TEXTLIST S4_Alarms
  0 = 'Station 4 Clamp A1 Failed to Advance... Check Q1.0...' | German: 'S4 0 Row 1 Failed To Advance.. Check Qxxx.x German' | French: 'S4 0 Row 1 Failed To Advance.. Check Qxxx.x French' | 汉语: '汉语'
  1 = 'Station 4 Clamp A1 Failed to Return... Check Q1.1...' | German: 'S4 1 Row 1 Failed To Return.. Check Qxxx.x German' | French: 'S4 1 Row 1 Failed To Return.. Check Qxxx.x French' | 汉语: '汉语'
  2 = 'Station 4 Clamp A1 Lost Advanced... Check I1.0...' | German: 'S4 2 Row 1 Lost Advance Position... Check Ixxx.x German' | French: 'S4 2 Row 1 Lost Advance Position... Check Ixxx.x French' | 汉语: '汉语'
  3 = 'Station 4 Clamp A1 Lost Returned... Check I1.1...' | German: 'S4 3 Row 1 Lost Return Position... Check Ixxx.x German' | French: 'S4 3 Row 1 Lost Return Position... Check Ixxx.x French'
  4 = 'Station 4 Clamp A1 Switch Fault... Check I1.0, I1.1...' | German: 'S4 4 Row 1 Switch Fault... Check Ixxx.x / Ixxx.x German' | French: 'S4 4 Row 1 Switch Fault... Check Ixxx.x / Ixxx.x French'
  5 = 'Spare' | German: 'S4 5 Row 1 Spare Message German' | French: 'S4 5 Row 1 Spare Message French'
  6 = 'Spare' | German: 'S4 6 Row 1 Spare Message German' | French: 'S4 6 Row 1 Spare Message French'
  7 = 'Spare' | German: 'S4 7 Row 1 Spare Message German' | French: 'S4 7 Row 1 Spare Message French'
  8 = 'Spare' | German: 'S4 8 Row 1 Spare Message German' | French: 'S4 8 Row 1 Spare Message French'
  9 = 'Spare' | German: 'S4 9 Row 1 Spare Message German' | French: 'S4 9 Row 1 Spare Message French'
  10 = 'Lock Cylinder A2 Failed to Lock... Check Q1.2...' | German: 'S4 10 Row 2 Failed To Advance.. Check Qxxx.x German' | French: 'S4 10 Row 2 Failed To Advance.. Check Qxxx.x French'
  11 = 'Lock Cylinder A2 Failed to Unlock... Check Q1.3...' | German: 'S4 11 Row 2 Failed To Return.. Check Qxxx.x German' | French: 'S4 11 Row 2 Failed To Return.. Check Qxxx.x French'
  12 = 'Lock Cylinder A2 Lost Locked... Check I1.2...' | German: 'S4 12 Row 2 Lost Advance Position... Check Ixxx.x German' | French: 'S4 12 Row 2 Lost Advance Position... Check Ixxx.x French'
  13 = 'Lock Cylinder A2 Lost Unlocked... Check I1.3...' | German: 'S4 13 Row 2 Lost Return Position... Check Ixxx.x German' | French: 'S4 13 Row 2 Lost Return Position... Check Ixxx.x French'
  14 = 'Lock Cylinder A2 Switch Fault... Check I1.2, I1.3...' | German: 'S4 14 Row 2 Switch Fault... Check Ixxx.x / Ixxx.x German' | French: 'S4 14 Row 2 Switch Fault... Check Ixxx.x / Ixxx.x French'
  15 = 'Spare' | German: 'S4 15 Row 2 Spare Message German' | French: 'S4 15 Row 2 Spare Message French'
  16 = 'Spare' | German: 'S4 16 Row 2 Spare Message German' | French: 'S4 16 Row 2 Spare Message French'
  17 = 'Spare' | German: 'S4 17 Row 2 Spare Message German' | French: 'S4 17 Row 2 Spare Message French'
  18 = 'Spare' | German: 'S4 18 Row 2 Spare Message German' | French: 'S4 18 Row 2 Spare Message French'
  19 = 'Spare' | German: 'S4 19 Row 2 Spare Message German' | French: 'S4 19 Row 2 Spare Message French'
  20 = 'Urger Cylinder A3 Failed to Urge... Check Q1.4...' | German: 'S4 20 Row 3 Failed To Advance.. Check Qxxx.x German' | French: 'S4 20 Row 3 Failed To Advance.. Check Qxxx.x French'
  21 = 'Urger Cylinder A3 Failed to Return... Check Q1.5...' | German: 'S4 21 Row 3 Failed To Return.. Check Qxxx.x German' | French: 'S4 21 Row 3 Failed To Return.. Check Qxxx.x French'
  22 = 'Urger Cylinder A3 Lost Urged... Check I1.4...' | German: 'S4 22 Row 3 Lost Advance Position... Check Ixxx.x German' | French: 'S4 22 Row 3 Lost Advance Position... Check Ixxx.x French'
  23 = 'Urger Cylinder A3 Lost Returned... Check I1.5...' | German: 'S4 23 Row 3 Lost Return Position... Check Ixxx.x German' | French: 'S4 23 Row 3 Lost Return Position... Check Ixxx.x French'
  24 = 'Urger Cylinder A3 Switch Fault... Check I1.4, I1.5...' | German: 'S4 24 Row 3 Switch Fault... Check Ixxx.x / Ixxx.x German' | French: 'S4 24 Row 3 Switch Fault... Check Ixxx.x / Ixxx.x French'
  25 = 'Spare' | German: 'S4 25 Row 3 Spare Message German' | French: 'S4 25 Row 3 Spare Message French'
  26 = 'Spare' | German: 'S4 26 Row 3 Spare Message German' | French: 'S4 26 Row 3 Spare Message French'
  27 = 'Spare' | German: 'S4 27 Row 3 Spare Message German' | French: 'S4 27 Row 3 Spare Message French'
  28 = 'Spare' | German: 'S4 28 Row 3 Spare Message German' | French: 'S4 28 Row 3 Spare Message French'
  29 = 'Spare' | German: 'S4 29 Row 3 Spare Message German' | French: 'S4 29 Row 3 Spare Message French'
  30 = 'Clamp Cylinder A1 Failed to Advance... Check Q1.0...' | German: 'S4 30 Row 4 Failed To Advance.. Check Qxxx.x German' | French: 'S4 30 Row 4 Failed To Advance.. Check Qxxx.x French'
  31 = 'Clamp Cylinder A1 Failed to Return... Check Q1.1...' | German: 'S4 31 Row 4 Failed To Return.. Check Qxxx.x German' | French: 'S4 31 Row 4 Failed To Return.. Check Qxxx.x French'
  32 = 'Clamp Cylinder A1 Lost Advanced... Check I1.0...' | German: 'S4 32 Row 4 Lost Advance Position... Check Ixxx.x German' | French: 'S4 32 Row 4 Lost Advance Position... Check Ixxx.x French'
  33 = 'Clamp Cylinder A1 Lost Returned... Check I1.1...' | German: 'S4 33 Row 4 Lost Return Position... Check Ixxx.x German' | French: 'S4 33 Row 4 Lost Return Position... Check Ixxx.x French'
  34 = 'Clamp Cylinder A1 Switch Fault... Check I1.0, I1.1...' | German: 'S4 34 Row 4 Switch Fault... Check Ixxx.x / Ixxx.x German' | French: 'S4 34 Row 4 Switch Fault... Check Ixxx.x / Ixxx.x French'
  35 = 'Spare' | German: 'S4 35 Row 4 Spare Message German' | French: 'S4 35 Row 4 Spare Message French'
  36 = 'Spare' | German: 'S4 36 Row 4 Spare Message German' | French: 'S4 36 Row 4 Spare Message French'
  37 = 'Spare' | German: 'S4 37 Row 4 Spare Message German' | French: 'S4 37 Row 4 Spare Message French'
  38 = 'Spare' | German: 'S4 38 Row 4 Spare Message German' | French: 'S4 38 Row 4 Spare Message French'
  39 = 'Spare' | German: 'S4 39 Row 4 Spare Message German' | French: 'S4 39 Row 4 Spare Message French'
  40 = 'Clamp Cylinder A1 Failed to Advance... Check Q1.0...' | German: 'S4 40 Row 5 Failed To Advance.. Check Qxxx.x German' | French: 'S4 40 Row 5 Failed To Advance.. Check Qxxx.x French'
  41 = 'Clamp Cylinder A1 Failed to Return... Check Q1.1...' | German: 'S4 41 Row 5 Failed To Return.. Check Qxxx.x German' | French: 'S4 41 Row 5 Failed To Return.. Check Qxxx.x French'
  42 = 'Clamp Cylinder A1 Lost Advanced... Check I1.0...' | German: 'S4 42 Row 5 Lost Advance Position... Check Ixxx.x German' | French: 'S4 42 Row 5 Lost Advance Position... Check Ixxx.x French'
  43 = 'Clamp Cylinder A1 Lost Returned... Check I1.1...' | German: 'S4 43 Row 5 Lost Return Position... Check Ixxx.x German' | French: 'S4 43 Row 5 Lost Return Position... Check Ixxx.x French'
  44 = 'Clamp Cylinder A1 Switch Fault... Check I1.0, I1.1...' | German: 'S4 44 Row 5 Switch Fault... Check Ixxx.x / Ixxx.x German' | French: 'S4 44 Row 5 Switch Fault... Check Ixxx.x / Ixxx.x French'
  45 = 'Spare' | German: 'S4 45 Row 5 Spare Message German' | French: 'S4 45 Row 5 Spare Message French'
  46 = 'Spare' | German: 'S4 46 Row 5 Spare Message German' | French: 'S4 46 Row 5 Spare Message French'
  47 = 'Spare' | German: 'S4 47 Row 5 Spare Message German' | French: 'S4 47 Row 5 Spare Message French'
  48 = 'Spare' | German: 'S4 48 Row 5 Spare Message German' | French: 'S4 48 Row 5 Spare Message French'
  49 = 'Spare' | German: 'S4 49 Row 5 Spare Message German' | French: 'S4 49 Row 5 Spare Message French'
  50 = 'Clamp Cylinder A1 Failed to Advance... Check Q1.0...' | German: 'S4 50 Row 6 Failed To Advance.. Check Qxxx.x German' | French: 'S4 50 Row 6 Failed To Advance.. Check Qxxx.x French'
  51 = 'Clamp Cylinder A1 Failed to Return... Check Q1.1...' | German: 'S4 51 Row 6 Failed To Return.. Check Qxxx.x German' | French: 'S4 51 Row 6 Failed To Return.. Check Qxxx.x French'
  52 = 'Clamp Cylinder A1 Lost Advanced... Check I1.0...' | German: 'S4 52 Row 6 Lost Advance Position... Check Ixxx.x German' | French: 'S4 52 Row 6 Lost Advance Position... Check Ixxx.x French'
  53 = 'Clamp Cylinder A1 Lost Returned... Check I1.1...' | German: 'S4 53 Row 6 Lost Return Position... Check Ixxx.x German' | French: 'S4 53 Row 6 Lost Return Position... Check Ixxx.x French'
  54 = 'Clamp Cylinder A1 Switch Fault... Check I1.0, I1.1...' | German: 'S4 54 Row 6 Switch Fault... Check Ixxx.x / Ixxx.x German' | French: 'S4 54 Row 6 Switch Fault... Check Ixxx.x / Ixxx.x French'
  55 = 'Spare' | German: 'S4 55 Row 6 Spare Message German' | French: 'S4 55 Row 6 Spare Message French'
  56 = 'Spare' | German: 'S4 56 Row 6 Spare Message German' | French: 'S4 56 Row 6 Spare Message French'
  57 = 'Spare' | German: 'S4 57 Row 6 Spare Message German' | French: 'S4 57 Row 6 Spare Message French'
  58 = 'Spare' | German: 'S4 58 Row 6 Spare Message German' | French: 'S4 58 Row 6 Spare Message French'
  59 = 'Spare' | German: 'S4 59 Row 6 Spare Message German' | French: 'S4 59 Row 6 Spare Message French'
  60 = 'Clamp Cylinder A1 Failed to Advance... Check Q1.0...' | German: 'S4 60 Row 7 Failed To Advance.. Check Qxxx.x German' | French: 'S4 60 Row 7 Failed To Advance.. Check Qxxx.x French'
  61 = 'Clamp Cylinder A1 Failed to Return... Check Q1.1...' | German: 'S4 61 Row 7 Failed To Return.. Check Qxxx.x German' | French: 'S4 61 Row 7 Failed To Return.. Check Qxxx.x French'
  62 = 'Clamp Cylinder A1 Lost Advanced... Check I1.0...' | German: 'S4 62 Row 7 Lost Advance Position... Check Ixxx.x German' | French: 'S4 62 Row 7 Lost Advance Position... Check Ixxx.x French'
  63 = 'Clamp Cylinder A1 Lost Returned... Check I1.1...' | German: 'S4 63 Row 7 Lost Return Position... Check Ixxx.x German' | French: 'S4 63 Row 7 Lost Return Position... Check Ixxx.x French'
  64 = 'Clamp Cylinder A1 Switch Fault... Check I1.0, I1.1...' | German: 'S4 64 Row 7 Switch Fault... Check Ixxx.x / Ixxx.x German' | French: 'S4 64 Row 7 Switch Fault... Check Ixxx.x / Ixxx.x French'
  65 = 'Spare' | German: 'S4 65 Row 7 Spare Message German' | French: 'S4 65 Row 7 Spare Message French'
  66 = 'Spare' | German: 'S4 66 Row 7 Spare Message German' | French: 'S4 66 Row 7 Spare Message French'
  67 = 'Spare' | German: 'S4 67 Row 7 Spare Message German' | French: 'S4 67 Row 7 Spare Message French'
  68 = 'Spare' | German: 'S4 68 Row 7 Spare Message German' | French: 'S4 68 Row 7 Spare Message French'
  69 = 'Spare' | German: 'S4 69 Row 7 Spare Message German' | French: 'S4 69 Row 7 Spare Message French'
  70 = 'Clamp Cylinder A1 Failed to Advance... Check Q1.0...' | German: 'S4 70 Row 8 Failed To Advance.. Check Qxxx.x German' | French: 'S4 70 Row 8 Failed To Advance.. Check Qxxx.x French'
  71 = 'Clamp Cylinder A1 Failed to Return... Check Q1.1...' | German: 'S4 71 Row 8 Failed To Return.. Check Qxxx.x German' | French: 'S4 71 Row 8 Failed To Return.. Check Qxxx.x French'
  72 = 'Clamp Cylinder A1 Lost Advanced... Check I1.0...' | German: 'S4 72 Row 8 Lost Advance Position... Check Ixxx.x German' | French: 'S4 72 Row 8 Lost Advance Position... Check Ixxx.x French'
  73 = 'Clamp Cylinder A1 Lost Returned... Check I1.1...' | German: 'S4 73 Row 8 Lost Return Position... Check Ixxx.x German' | French: 'S4 73 Row 8 Lost Return Position... Check Ixxx.x French'
  74 = 'Clamp Cylinder A1 Switch Fault... Check I1.0, I1.1...' | German: 'S4 74 Row 8 Switch Fault... Check Ixxx.x / Ixxx.x German' | French: 'S4 74 Row 8 Switch Fault... Check Ixxx.x / Ixxx.x French'
  75 = 'Spare' | German: 'S4 75 Row 8 Spare Message German' | French: 'S4 75 Row 8 Spare Message French'
  76 = 'Spare' | German: 'S4 76 Row 8 Spare Message German' | French: 'S4 76 Row 8 Spare Message French'
  77 = 'Spare' | German: 'S4 77 Row 8 Spare Message German' | French: 'S4 77 Row 8 Spare Message French'
  78 = 'Spare' | German: 'S4 78 Row 8 Spare Message German' | French: 'S4 78 Row 8 Spare Message French'
  79 = 'Spare' | German: 'S4 79 Row 8 Spare Message German' | French: 'S4 79 Row 8 Spare Message French'
  80 = 'Clamp Cylinder A1 Failed to Advance... Check Q1.0...' | German: 'S4 80 Row 9 Failed To Advance.. Check Qxxx.x German' | French: 'S4 80 Row 9 Failed To Advance.. Check Qxxx.x French'
  81 = 'Clamp Cylinder A1 Failed to Return... Check Q1.1...' | German: 'S4 81 Row 9 Failed To Return.. Check Qxxx.x German' | French: 'S4 81 Row 9 Failed To Return.. Check Qxxx.x French'
  82 = 'Clamp Cylinder A1 Lost Advanced... Check I1.0...' | German: 'S4 82 Row 9 Lost Advance Position... Check Ixxx.x German' | French: 'S4 82 Row 9 Lost Advance Position... Check Ixxx.x French'
  83 = 'Clamp Cylinder A1 Lost Returned... Check I1.1...' | German: 'S4 83 Row 9 Lost Return Position... Check Ixxx.x German' | French: 'S4 83 Row 9 Lost Return Position... Check Ixxx.x French'
  84 = 'Clamp Cylinder A1 Switch Fault... Check I1.0, I1.1...' | German: 'S4 84 Row 9 Switch Fault... Check Ixxx.x / Ixxx.x German' | French: 'S4 84 Row 9 Switch Fault... Check Ixxx.x / Ixxx.x French'
  85 = 'Spare' | German: 'S4 85 Row 9 Spare Message German' | French: 'S4 85 Row 9 Spare Message French'
  86 = 'Spare' | German: 'S4 86 Row 9 Spare Message German' | French: 'S4 86 Row 9 Spare Message French'
  87 = 'Spare' | German: 'S4 87 Row 9 Spare Message German' | French: 'S4 87 Row 9 Spare Message French'
  88 = 'Spare' | German: 'S4 88 Row 9 Spare Message German' | French: 'S4 88 Row 9 Spare Message French'
  89 = 'Spare' | German: 'S4 89 Row 9 Spare Message German' | French: 'S4 89 Row 9 Spare Message French'
  90 = 'Clamp Cylinder A1 Failed to Advance... Check Q1.0...' | German: 'S4 90 Row 10 Failed To Advance.. Check Qxxx.x German' | French: 'S4 90 Row 10 Failed To Advance.. Check Qxxx.x French'
  91 = 'Clamp Cylinder A1 Failed to Return... Check Q1.1...' | German: 'S4 91 Row 10 Failed To Return.. Check Qxxx.x German' | French: 'S4 91 Row 10 Failed To Return.. Check Qxxx.x French'
  92 = 'Clamp Cylinder A1 Lost Advanced... Check I1.0...' | German: 'S4 92 Row 10 Lost Advance Position... Check Ixxx.x German' | French: 'S4 92 Row 10 Lost Advance Position... Check Ixxx.x French'
  93 = 'Clamp Cylinder A1 Lost Returned... Check I1.1...' | German: 'S4 93 Row 10 Lost Return Position... Check Ixxx.x German' | French: 'S4 93 Row 10 Lost Return Position... Check Ixxx.x French'
  94 = 'Clamp Cylinder A1 Switch Fault... Check I1.0, I1.1...' | German: 'S4 94 Row 10 Switch Fault... Check Ixxx.x / Ixxx.x German' | French: 'S4 94 Row 10 Switch Fault... Check Ixxx.x / Ixxx.x French'
  95 = 'Spare' | German: 'S4 95 Row 10 Spare Message German' | French: 'S4 95 Row 10 Spare Message French'
  96 = 'Spare' | German: 'S4 96 Row 10 Spare Message German' | French: 'S4 96 Row 10 Spare Message French'
  97 = 'Spare' | German: 'S4 97 Row 10 Spare Message German' | French: 'S4 97 Row 10 Spare Message French'
  98 = 'Spare' | German: 'S4 98 Row 10 Spare Message German' | French: 'S4 98 Row 10 Spare Message French'
  99 = 'Spare' | German: 'S4 99 Row 10 Spare Message German' | French: 'S4 99 Row 10 Spare Message French'
  100 = 'Clamp Cylinder A1 Failed to Advance... Check Q1.0...' | German: 'S4 100 Row 11 Failed To Advance.. Check Qxxx.x German' | French: 'S4 100 Row 11 Failed To Advance.. Check Qxxx.x French'
  101 = 'Clamp Cylinder A1 Failed to Return... Check Q1.1...' | German: 'S4 101 Row 11 Failed To Return.. Check Qxxx.x German' | French: 'S4 101 Row 11 Failed To Return.. Check Qxxx.x French'
  102 = 'Clamp Cylinder A1 Lost Advanced... Check I1.0...' | German: 'S4 102 Row 11 Lost Advance Position... Check Ixxx.x German' | French: 'S4 102 Row 11 Lost Advance Position... Check Ixxx.x French'
  103 = 'Clamp Cylinder A1 Lost Returned... Check I1.1...' | German: 'S4 103 Row 11 Lost Return Position... Check Ixxx.x German' | French: 'S4 103 Row 11 Lost Return Position... Check Ixxx.x French'
  104 = 'Clamp Cylinder A1 Switch Fault... Check I1.0, I1.1...' | German: 'S4 104 Row 11 Switch Fault... Check Ixxx.x / Ixxx.x German' | French: 'S4 104 Row 11 Switch Fault... Check Ixxx.x / Ixxx.x French'
  105 = 'Spare' | German: 'S4 105 Row 11 Spare Message German' | French: 'S4 105 Row 11 Spare Message French'
  106 = 'Spare' | German: 'S4 106 Row 11 Spare Message German' | French: 'S4 106 Row 11 Spare Message French'
  107 = 'Spare' | German: 'S4 107 Row 11 Spare Message German' | French: 'S4 107 Row 11 Spare Message French'
  108 = 'Spare' | German: 'S4 108 Row 11 Spare Message German' | French: 'S4 108 Row 11 Spare Message French'
  109 = 'Spare' | German: 'S4 109 Row 11 Spare Message German' | French: 'S4 109 Row 11 Spare Message French'
  110 = 'Clamp Cylinder A1 Failed to Advance... Check Q1.0...' | German: 'S4 110 Row 12 Failed To Advance.. Check Qxxx.x German' | French: 'S4 110 Row 12 Failed To Advance.. Check Qxxx.x French'
  111 = 'Clamp Cylinder A1 Failed to Return... Check Q1.1...' | German: 'S4 111 Row 12 Failed To Return.. Check Qxxx.x German' | French: 'S4 111 Row 12 Failed To Return.. Check Qxxx.x French'
  112 = 'Clamp Cylinder A1 Lost Advanced... Check I1.0...' | German: 'S4 112 Row 12 Lost Advance Position... Check Ixxx.x German' | French: 'S4 112 Row 12 Lost Advance Position... Check Ixxx.x French'
  113 = 'Clamp Cylinder A1 Lost Returned... Check I1.1...' | German: 'S4 113 Row 12 Lost Return Position... Check Ixxx.x German' | French: 'S4 113 Row 12 Lost Return Position... Check Ixxx.x French'
  114 = 'Clamp Cylinder A1 Switch Fault... Check I1.0, I1.1...' | German: 'S4 114 Row 12 Switch Fault... Check Ixxx.x / Ixxx.x German' | French: 'S4 114 Row 12 Switch Fault... Check Ixxx.x / Ixxx.x French'
  115 = 'Spare' | German: 'S4 115 Row 12 Spare Message German' | French: 'S4 115 Row 12 Spare Message French'
  116 = 'Spare' | German: 'S4 116 Row 12 Spare Message German' | French: 'S4 116 Row 12 Spare Message French'
  117 = 'Spare' | German: 'S4 117 Row 12 Spare Message German' | French: 'S4 117 Row 12 Spare Message French'
  118 = 'Spare' | German: 'S4 118 Row 12 Spare Message German' | French: 'S4 118 Row 12 Spare Message French'
  119 = 'Spare' | German: 'S4 119 Row 12 Spare Message German' | French: 'S4 119 Row 12 Spare Message French'
  120 = 'Clamp Cylinder A1 Failed to Advance... Check Q1.0...' | German: 'S4 120 Row 13 Failed To Advance.. Check Qxxx.x German' | French: 'S4 120 Row 13 Failed To Advance.. Check Qxxx.x French'
  121 = 'Clamp Cylinder A1 Failed to Return... Check Q1.1...' | German: 'S4 121 Row 13 Failed To Return.. Check Qxxx.x German' | French: 'S4 121 Row 13 Failed To Return.. Check Qxxx.x French'
  122 = 'Clamp Cylinder A1 Lost Advanced... Check I1.0...' | German: 'S4 122 Row 13 Lost Advance Position... Check Ixxx.x German' | French: 'S4 122 Row 13 Lost Advance Position... Check Ixxx.x French'
  123 = 'Clamp Cylinder A1 Lost Returned... Check I1.1...' | German: 'S4 123 Row 13 Lost Return Position... Check Ixxx.x German' | French: 'S4 123 Row 13 Lost Return Position... Check Ixxx.x French'
  124 = 'Clamp Cylinder A1 Switch Fault... Check I1.0, I1.1...' | German: 'S4 124 Row 13 Switch Fault... Check Ixxx.x / Ixxx.x German' | French: 'S4 124 Row 13 Switch Fault... Check Ixxx.x / Ixxx.x French'
  125 = 'Spare' | German: 'S4 125 Row 13 Spare Message German' | French: 'S4 125 Row 13 Spare Message French'
  126 = 'Spare' | German: 'S4 126 Row 13 Spare Message German' | French: 'S4 126 Row 13 Spare Message French'
  127 = 'Spare' | German: 'S4 127 Row 13 Spare Message German' | French: 'S4 127 Row 13 Spare Message French'
  128 = 'Spare' | German: 'S4 128 Row 13 Spare Message German' | French: 'S4 128 Row 13 Spare Message French'
  129 = 'Spare' | German: 'S4 129 Row 13 Spare Message German' | French: 'S4 129 Row 13 Spare Message French'
  130 = 'Clamp Cylinder A1 Failed to Advance... Check Q1.0...' | German: 'S4 130 Row 14 Failed To Advance.. Check Qxxx.x German' | French: 'S4 130 Row 14 Failed To Advance.. Check Qxxx.x French'
  131 = 'Clamp Cylinder A1 Failed to Return... Check Q1.1...' | German: 'S4 131 Row 14 Failed To Return.. Check Qxxx.x German' | French: 'S4 131 Row 14 Failed To Return.. Check Qxxx.x French'
  132 = 'Clamp Cylinder A1 Lost Advanced... Check I1.0...' | German: 'S4 132 Row 14 Lost Advance Position... Check Ixxx.x German' | French: 'S4 132 Row 14 Lost Advance Position... Check Ixxx.x French'
  133 = 'Clamp Cylinder A1 Lost Returned... Check I1.1...' | German: 'S4 133 Row 14 Lost Return Position... Check Ixxx.x German' | French: 'S4 133 Row 14 Lost Return Position... Check Ixxx.x French'
  134 = 'Clamp Cylinder A1 Switch Fault... Check I1.0, I1.1...' | German: 'S4 134 Row 14 Switch Fault... Check Ixxx.x / Ixxx.x German' | French: 'S4 134 Row 14 Switch Fault... Check Ixxx.x / Ixxx.x French'
  135 = 'Spare' | German: 'S4 135 Row 14 Spare Message German' | French: 'S4 135 Row 14 Spare Message French'
  136 = 'Spare' | German: 'S4 136 Row 14 Spare Message German' | French: 'S4 136 Row 14 Spare Message French'
  137 = 'Spare' | German: 'S4 137 Row 14 Spare Message German' | French: 'S4 137 Row 14 Spare Message French'
  138 = 'Spare' | German: 'S4 138 Row 14 Spare Message German' | French: 'S4 138 Row 14 Spare Message French'
  139 = 'Spare' | German: 'S4 139 Row 14 Spare Message German' | French: 'S4 139 Row 14 Spare Message French'
  140 = 'Clamp Cylinder A1 Failed to Advance... Check Q1.0...' | German: 'S4 140 Row 15 Failed To Advance.. Check Qxxx.x German' | French: 'S4 140 Row 15 Failed To Advance.. Check Qxxx.x French'
  141 = 'Clamp Cylinder A1 Failed to Return... Check Q1.1...' | German: 'S4 141 Row 15 Failed To Return.. Check Qxxx.x German' | French: 'S4 141 Row 15 Failed To Return.. Check Qxxx.x French'
  142 = 'Clamp Cylinder A1 Lost Advanced... Check I1.0...' | German: 'S4 142 Row 15 Lost Advance Position... Check Ixxx.x German' | French: 'S4 142 Row 15 Lost Advance Position... Check Ixxx.x French'
  143 = 'Clamp Cylinder A1 Lost Returned... Check I1.1...' | German: 'S4 143 Row 15 Lost Return Position... Check Ixxx.x German' | French: 'S4 143 Row 15 Lost Return Position... Check Ixxx.x French'
  144 = 'Clamp Cylinder A1 Switch Fault... Check I1.0, I1.1...' | German: 'S4 144 Row 15 Switch Fault... Check Ixxx.x / Ixxx.x German' | French: 'S4 144 Row 15 Switch Fault... Check Ixxx.x / Ixxx.x French'
  145 = 'Spare' | German: 'S4 145 Row 15 Spare Message German' | French: 'S4 145 Row 15 Spare Message French'
  146 = 'Spare' | German: 'S4 146 Row 15 Spare Message German' | French: 'S4 146 Row 15 Spare Message French'
  147 = 'Spare' | German: 'S4 147 Row 15 Spare Message German' | French: 'S4 147 Row 15 Spare Message French'
  148 = 'Spare' | German: 'S4 148 Row 15 Spare Message German' | French: 'S4 148 Row 15 Spare Message French'
  149 = 'Spare' | German: 'S4 149 Row 15 Spare Message German' | French: 'S4 149 Row 15 Spare Message French'
  150 = 'Clamp Cylinder A1 Failed to Advance... Check Q1.0...' | German: 'S4 150 Row 16 Failed To Advance.. Check Qxxx.x German' | French: 'S4 150 Row 16 Failed To Advance.. Check Qxxx.x French'
  151 = 'Clamp Cylinder A1 Failed to Return... Check Q1.1...' | German: 'S4 151 Row 16 Failed To Return.. Check Qxxx.x German' | French: 'S4 151 Row 16 Failed To Return.. Check Qxxx.x French'
  152 = 'Clamp Cylinder A1 Lost Advanced... Check I1.0...' | German: 'S4 152 Row 16 Lost Advance Position... Check Ixxx.x German' | French: 'S4 152 Row 16 Lost Advance Position... Check Ixxx.x French'
  153 = 'Clamp Cylinder A1 Lost Returned... Check I1.1...' | German: 'S4 153 Row 16 Lost Return Position... Check Ixxx.x German' | French: 'S4 153 Row 16 Lost Return Position... Check Ixxx.x French'
  154 = 'Clamp Cylinder A1 Switch Fault... Check I1.0, I1.1...' | German: 'S4 154 Row 16 Switch Fault... Check Ixxx.x / Ixxx.x German' | French: 'S4 154 Row 16 Switch Fault... Check Ixxx.x / Ixxx.x French'
  155 = 'Spare' | German: 'S4 155 Row 16 Spare Message German' | French: 'S4 155 Row 16 Spare Message French'
  156 = 'Spare' | German: 'S4 156 Row 16 Spare Message German' | French: 'S4 156 Row 16 Spare Message French'
  157 = 'Spare' | German: 'S4 157 Row 16 Spare Message German' | French: 'S4 157 Row 16 Spare Message French'
  158 = 'Spare' | German: 'S4 158 Row 16 Spare Message German' | French: 'S4 158 Row 16 Spare Message French'
  159 = 'Spare' | German: 'S4 159 Row 16 Spare Message German' | French: 'S4 159 Row 16 Spare Message French'
  160 = 'Clamp Cylinder A1 Failed to Advance... Check Q1.0...' | German: 'S4 160 Row 17 Failed To Advance.. Check Qxxx.x German' | French: 'S4 160 Row 17 Failed To Advance.. Check Qxxx.x French'
  161 = 'Clamp Cylinder A1 Failed to Return... Check Q1.1...' | German: 'S4 161 Row 17 Failed To Return.. Check Qxxx.x German' | French: 'S4 161 Row 17 Failed To Return.. Check Qxxx.x French'
  162 = 'Clamp Cylinder A1 Lost Advanced... Check I1.0...' | German: 'S4 162 Row 17 Lost Advance Position... Check Ixxx.x German' | French: 'S4 162 Row 17 Lost Advance Position... Check Ixxx.x French'
  163 = 'Clamp Cylinder A1 Lost Returned... Check I1.1...' | German: 'S4 163 Row 17 Lost Return Position... Check Ixxx.x German' | French: 'S4 163 Row 17 Lost Return Position... Check Ixxx.x French'
  164 = 'Clamp Cylinder A1 Switch Fault... Check I1.0, I1.1...' | German: 'S4 164 Row 17 Switch Fault... Check Ixxx.x / Ixxx.x German' | French: 'S4 164 Row 17 Switch Fault... Check Ixxx.x / Ixxx.x French'
  165 = 'Spare' | German: 'S4 165 Row 17 Spare Message German' | French: 'S4 165 Row 17 Spare Message French'
  166 = 'Spare' | German: 'S4 166 Row 17 Spare Message German' | French: 'S4 166 Row 17 Spare Message French'
  167 = 'Spare' | German: 'S4 167 Row 17 Spare Message German' | French: 'S4 167 Row 17 Spare Message French'
  168 = 'Spare' | German: 'S4 168 Row 17 Spare Message German' | French: 'S4 168 Row 17 Spare Message French'
  169 = 'Spare' | German: 'S4 169 Row 17 Spare Message German' | French: 'S4 169 Row 17 Spare Message French'
  170 = 'Clamp Cylinder A1 Failed to Advance... Check Q1.0...' | German: 'S4 170 Row 18 Failed To Advance.. Check Qxxx.x German' | French: 'S4 170 Row 18 Failed To Advance.. Check Qxxx.x French'
  171 = 'Clamp Cylinder A1 Failed to Return... Check Q1.1...' | German: 'S4 171 Row 18 Failed To Return.. Check Qxxx.x German' | French: 'S4 171 Row 18 Failed To Return.. Check Qxxx.x French'
  172 = 'Clamp Cylinder A1 Lost Advanced... Check I1.0...' | German: 'S4 172 Row 18 Lost Advance Position... Check Ixxx.x German' | French: 'S4 172 Row 18 Lost Advance Position... Check Ixxx.x French'
  173 = 'Clamp Cylinder A1 Lost Returned... Check I1.1...' | German: 'S4 173 Row 18 Lost Return Position... Check Ixxx.x German' | French: 'S4 173 Row 18 Lost Return Position... Check Ixxx.x French'
  174 = 'Clamp Cylinder A1 Switch Fault... Check I1.0, I1.1...' | German: 'S4 174 Row 18 Switch Fault... Check Ixxx.x / Ixxx.x German' | French: 'S4 174 Row 18 Switch Fault... Check Ixxx.x / Ixxx.x French'
  175 = 'Spare' | German: 'S4 175 Row 18 Spare Message German' | French: 'S4 175 Row 18 Spare Message French'
  176 = 'Spare' | German: 'S4 176 Row 18 Spare Message German' | French: 'S4 176 Row 18 Spare Message French'
  177 = 'Spare' | German: 'S4 177 Row 18 Spare Message German' | French: 'S4 177 Row 18 Spare Message French'
  178 = 'Spare' | German: 'S4 178 Row 18 Spare Message German' | French: 'S4 178 Row 18 Spare Message French'
  179 = 'Spare' | German: 'S4 179 Row 18 Spare Message German' | French: 'S4 179 Row 18 Spare Message French'
  180 = 'Clamp Cylinder A1 Failed to Advance... Check Q1.0...' | German: 'S4 180 Row 19 Failed To Advance.. Check Qxxx.x German' | French: 'S4 180 Row 19 Failed To Advance.. Check Qxxx.x French'
  181 = 'Clamp Cylinder A1 Failed to Return... Check Q1.1...' | German: 'S4 181 Row 19 Failed To Return.. Check Qxxx.x German' | French: 'S4 181 Row 19 Failed To Return.. Check Qxxx.x French'
  182 = 'Clamp Cylinder A1 Lost Advanced... Check I1.0...' | German: 'S4 182 Row 19 Lost Advance Position... Check Ixxx.x German' | French: 'S4 182 Row 19 Lost Advance Position... Check Ixxx.x French'
  183 = 'Clamp Cylinder A1 Lost Returned... Check I1.1...' | German: 'S4 183 Row 19 Lost Return Position... Check Ixxx.x German' | French: 'S4 183 Row 19 Lost Return Position... Check Ixxx.x French'
  184 = 'Clamp Cylinder A1 Switch Fault... Check I1.0, I1.1...' | German: 'S4 184 Row 19 Switch Fault... Check Ixxx.x / Ixxx.x German' | French: 'S4 184 Row 19 Switch Fault... Check Ixxx.x / Ixxx.x French'
  185 = 'Spare' | German: 'S4 185 Row 19 Spare Message German' | French: 'S4 185 Row 19 Spare Message French'
  186 = 'Spare' | German: 'S4 186 Row 19 Spare Message German' | French: 'S4 186 Row 19 Spare Message French'
  187 = 'Spare' | German: 'S4 187 Row 19 Spare Message German' | French: 'S4 187 Row 19 Spare Message French'
  188 = 'Spare' | German: 'S4 188 Row 19 Spare Message German' | French: 'S4 188 Row 19 Spare Message French'
  189 = 'Spare' | German: 'S4 189 Row 19 Spare Message German' | French: 'S4 189 Row 19 Spare Message French'
  190 = 'Clamp Cylinder A1 Failed to Advance... Check Q1.0...' | German: 'S4 190 Row 20 Failed To Advance.. Check Qxxx.x German' | French: 'S4 190 Row 20 Failed To Advance.. Check Qxxx.x French'
  191 = 'Clamp Cylinder A1 Failed to Return... Check Q1.1...' | German: 'S4 191 Row 20 Failed To Return.. Check Qxxx.x German' | French: 'S4 191 Row 20 Failed To Return.. Check Qxxx.x French'
  192 = 'Clamp Cylinder A1 Lost Advanced... Check I1.0...' | German: 'S4 192 Row 20 Lost Advance Position... Check Ixxx.x German' | French: 'S4 192 Row 20 Lost Advance Position... Check Ixxx.x French'
  193 = 'Clamp Cylinder A1 Lost Returned... Check I1.1...' | German: 'S4 193 Row 20 Lost Return Position... Check Ixxx.x German' | French: 'S4 193 Row 20 Lost Return Position... Check Ixxx.x French'
  194 = 'Clamp Cylinder A1 Switch Fault... Check I1.0, I1.1...' | German: 'S4 194 Row 20 Switch Fault... Check Ixxx.x / Ixxx.x German' | French: 'S4 194 Row 20 Switch Fault... Check Ixxx.x / Ixxx.x French'
  195 = 'Spare' | German: 'S4 195 Row 20 Spare Message German' | French: 'S4 195 Row 20 Spare Message French'
  196 = 'Spare' | German: 'S4 196 Row 20 Spare Message German' | French: 'S4 196 Row 20 Spare Message French'
  197 = 'Spare' | German: 'S4 197 Row 20 Spare Message German' | French: 'S4 197 Row 20 Spare Message French'
  198 = 'Spare' | German: 'S4 198 Row 20 Spare Message German' | French: 'S4 198 Row 20 Spare Message French'
  199 = 'Spare' | German: 'S4 199 Row 20 Spare Message German' | French: 'S4 199 Row 20 Spare Message French'
  200 = 'Clamp Cylinder A1 Failed to Advance... Check Q1.0...' | German: 'S4 200 Row 21 Failed To Advance.. Check Qxxx.x German' | French: 'S4 200 Row 21 Failed To Advance.. Check Qxxx.x French'
  201 = 'Clamp Cylinder A1 Failed to Return... Check Q1.1...' | German: 'S4 201 Row 21 Failed To Return.. Check Qxxx.x German' | French: 'S4 201 Row 21 Failed To Return.. Check Qxxx.x French'
  202 = 'Clamp Cylinder A1 Lost Advanced... Check I1.0...' | German: 'S4 202 Row 21 Lost Advance Position... Check Ixxx.x German' | French: 'S4 202 Row 21 Lost Advance Position... Check Ixxx.x French'
  203 = 'Clamp Cylinder A1 Lost Returned... Check I1.1...' | German: 'S4 203 Row 21 Lost Return Position... Check Ixxx.x German' | French: 'S4 203 Row 21 Lost Return Position... Check Ixxx.x French'
  204 = 'Clamp Cylinder A1 Switch Fault... Check I1.0, I1.1...' | German: 'S4 204 Row 21 Switch Fault... Check Ixxx.x / Ixxx.x German' | French: 'S4 204 Row 21 Switch Fault... Check Ixxx.x / Ixxx.x French'
  205 = 'Spare' | German: 'S4 205 Row 21 Spare Message German' | French: 'S4 205 Row 21 Spare Message French'
  206 = 'Spare' | German: 'S4 206 Row 21 Spare Message German' | French: 'S4 206 Row 21 Spare Message French'
  207 = 'Spare' | German: 'S4 207 Row 21 Spare Message German' | French: 'S4 207 Row 21 Spare Message French'
  208 = 'Spare' | German: 'S4 208 Row 21 Spare Message German' | French: 'S4 208 Row 21 Spare Message French'
  209 = 'Spare' | German: 'S4 209 Row 21 Spare Message German' | French: 'S4 209 Row 21 Spare Message French'
  210 = 'Clamp Cylinder A1 Failed to Advance... Check Q1.0...' | German: 'S4 210 Row 22 Failed To Advance.. Check Qxxx.x German' | French: 'S4 210 Row 22 Failed To Advance.. Check Qxxx.x French'
  211 = 'Clamp Cylinder A1 Failed to Return... Check Q1.1...' | German: 'S4 211 Row 22 Failed To Return.. Check Qxxx.x German' | French: 'S4 211 Row 22 Failed To Return.. Check Qxxx.x French'
  212 = 'Clamp Cylinder A1 Lost Advanced... Check I1.0...' | German: 'S4 212 Row 22 Lost Advance Position... Check Ixxx.x German' | French: 'S4 212 Row 22 Lost Advance Position... Check Ixxx.x French'
  213 = 'Clamp Cylinder A1 Lost Returned... Check I1.1...' | German: 'S4 213 Row 22 Lost Return Position... Check Ixxx.x German' | French: 'S4 213 Row 22 Lost Return Position... Check Ixxx.x French'
  214 = 'Clamp Cylinder A1 Switch Fault... Check I1.0, I1.1...' | German: 'S4 214 Row 22 Switch Fault... Check Ixxx.x / Ixxx.x German' | French: 'S4 214 Row 22 Switch Fault... Check Ixxx.x / Ixxx.x French'
  215 = 'Spare' | German: 'S4 215 Row 22 Spare Message German' | French: 'S4 215 Row 22 Spare Message French'
  216 = 'Spare' | German: 'S4 216 Row 22 Spare Message German' | French: 'S4 216 Row 22 Spare Message French'
  217 = 'Spare' | German: 'S4 217 Row 22 Spare Message German' | French: 'S4 217 Row 22 Spare Message French'
  218 = 'Spare' | German: 'S4 218 Row 22 Spare Message German' | French: 'S4 218 Row 22 Spare Message French'
  219 = 'Spare' | German: 'S4 219 Row 22 Spare Message German' | French: 'S4 219 Row 22 Spare Message French'
  220 = 'Clamp Cylinder A1 Failed to Advance... Check Q1.0...' | German: 'S4 220 Row 23 Failed To Advance.. Check Qxxx.x German' | French: 'S4 220 Row 23 Failed To Advance.. Check Qxxx.x French'
  221 = 'Clamp Cylinder A1 Failed to Return... Check Q1.1...' | German: 'S4 221 Row 23 Failed To Return.. Check Qxxx.x German' | French: 'S4 221 Row 23 Failed To Return.. Check Qxxx.x French'
  222 = 'Clamp Cylinder A1 Lost Advanced... Check I1.0...' | German: 'S4 222 Row 23 Lost Advance Position... Check Ixxx.x German' | French: 'S4 222 Row 23 Lost Advance Position... Check Ixxx.x French'
  223 = 'Clamp Cylinder A1 Lost Returned... Check I1.1...' | German: 'S4 223 Row 23 Lost Return Position... Check Ixxx.x German' | French: 'S4 223 Row 23 Lost Return Position... Check Ixxx.x French'
  224 = 'Clamp Cylinder A1 Switch Fault... Check I1.0, I1.1...' | German: 'S4 224 Row 23 Switch Fault... Check Ixxx.x / Ixxx.x German' | French: 'S4 224 Row 23 Switch Fault... Check Ixxx.x / Ixxx.x French'
  225 = 'Spare' | German: 'S4 225 Row 23 Spare Message German' | French: 'S4 225 Row 23 Spare Message French'
  226 = 'Spare' | German: 'S4 226 Row 23 Spare Message German' | French: 'S4 226 Row 23 Spare Message French'
  227 = 'Spare' | German: 'S4 227 Row 23 Spare Message German' | French: 'S4 227 Row 23 Spare Message French'
  228 = 'Spare' | German: 'S4 228 Row 23 Spare Message German' | French: 'S4 228 Row 23 Spare Message French'
  229 = 'Spare' | German: 'S4 229 Row 23 Spare Message German' | French: 'S4 229 Row 23 Spare Message French'
  230 = 'Clamp Cylinder A1 Failed to Advance... Check Q1.0...' | German: 'S4 230 Row 24 Failed To Advance.. Check Qxxx.x German' | French: 'S4 230 Row 24 Failed To Advance.. Check Qxxx.x French'
  231 = 'Clamp Cylinder A1 Failed to Return... Check Q1.1...' | German: 'S4 231 Row 24 Failed To Return.. Check Qxxx.x German' | French: 'S4 231 Row 24 Failed To Return.. Check Qxxx.x French'
  232 = 'Clamp Cylinder A1 Lost Advanced... Check I1.0...' | German: 'S4 232 Row 24 Lost Advance Position... Check Ixxx.x German' | French: 'S4 232 Row 24 Lost Advance Position... Check Ixxx.x French'
  233 = 'Clamp Cylinder A1 Lost Returned... Check I1.1...' | German: 'S4 233 Row 24 Lost Return Position... Check Ixxx.x German' | French: 'S4 233 Row 24 Lost Return Position... Check Ixxx.x French'
  234 = 'Clamp Cylinder A1 Switch Fault... Check I1.0, I1.1...' | German: 'S4 234 Row 24 Switch Fault... Check Ixxx.x / Ixxx.x German' | French: 'S4 234 Row 24 Switch Fault... Check Ixxx.x / Ixxx.x French'
  235 = 'Spare' | German: 'S4 235 Row 24 Spare Message German' | French: 'S4 235 Row 24 Spare Message French'
  236 = 'Spare' | German: 'S4 236 Row 24 Spare Message German' | French: 'S4 236 Row 24 Spare Message French'
  237 = 'Spare' | German: 'S4 237 Row 24 Spare Message German' | French: 'S4 237 Row 24 Spare Message French'
  238 = 'Spare' | German: 'S4 238 Row 24 Spare Message German' | French: 'S4 238 Row 24 Spare Message French'
  239 = 'Spare' | German: 'S4 239 Row 24 Spare Message German' | French: 'S4 239 Row 24 Spare Message French'
  240 = 'Clamp Cylinder A1 Failed to Advance... Check Q1.0...' | German: 'S4 240 Row 25 Failed To Advance.. Check Qxxx.x German' | French: 'S4 240 Row 25 Failed To Advance.. Check Qxxx.x French'
  241 = 'Clamp Cylinder A1 Failed to Return... Check Q1.1...' | German: 'S4 241 Row 25 Failed To Return.. Check Qxxx.x German' | French: 'S4 241 Row 25 Failed To Return.. Check Qxxx.x French'
  242 = 'Clamp Cylinder A1 Lost Advanced... Check I1.0...' | German: 'S4 242 Row 25 Lost Advance Position... Check Ixxx.x German' | French: 'S4 242 Row 25 Lost Advance Position... Check Ixxx.x French'
  243 = 'Clamp Cylinder A1 Lost Returned... Check I1.1...' | German: 'S4 243 Row 25 Lost Return Position... Check Ixxx.x German' | French: 'S4 243 Row 25 Lost Return Position... Check Ixxx.x French'
  244 = 'Clamp Cylinder A1 Switch Fault... Check I1.0, I1.1...' | German: 'S4 244 Row 25 Switch Fault... Check Ixxx.x / Ixxx.x German' | French: 'S4 244 Row 25 Switch Fault... Check Ixxx.x / Ixxx.x French'
  245 = 'Spare' | German: 'S4 245 Row 25 Spare Message German' | French: 'S4 245 Row 25 Spare Message French'
  246 = 'Spare' | German: 'S4 246 Row 25 Spare Message German' | French: 'S4 246 Row 25 Spare Message French'
  247 = 'Spare' | German: 'S4 247 Row 25 Spare Message German' | French: 'S4 247 Row 25 Spare Message French'
  248 = 'Spare' | German: 'S4 248 Row 25 Spare Message German' | French: 'S4 248 Row 25 Spare Message French'
  249 = 'Spare' | German: 'S4 249 Row 25 Spare Message German' | French: 'S4 249 Row 25 Spare Message French'
  250 = 'Clamp Cylinder A1 Failed to Advance... Check Q1.0...' | German: 'S4 250 Row 26 Failed To Advance.. Check Qxxx.x German' | French: 'S4 250 Row 26 Failed To Advance.. Check Qxxx.x French'
  251 = 'Clamp Cylinder A1 Failed to Return... Check Q1.1...' | German: 'S4 251 Row 26 Failed To Return.. Check Qxxx.x German' | French: 'S4 251 Row 26 Failed To Return.. Check Qxxx.x French'
  252 = 'Clamp Cylinder A1 Lost Advanced... Check I1.0...' | German: 'S4 252 Row 26 Lost Advance Position... Check Ixxx.x German' | French: 'S4 252 Row 26 Lost Advance Position... Check Ixxx.x French'
  253 = 'Clamp Cylinder A1 Lost Returned... Check I1.1...' | German: 'S4 253 Row 26 Lost Return Position... Check Ixxx.x German' | French: 'S4 253 Row 26 Lost Return Position... Check Ixxx.x French'
  254 = 'Clamp Cylinder A1 Switch Fault... Check I1.0, I1.1...' | German: 'S4 254 Row 26 Switch Fault... Check Ixxx.x / Ixxx.x German' | French: 'S4 254 Row 26 Switch Fault... Check Ixxx.x / Ixxx.x French'
  255 = 'Spare' | German: 'S4 255 Row 26 Spare Message German' | French: 'S4 255 Row 26 Spare Message French'
  256 = 'Spare' | German: 'S4 256 Row 26 Spare Message German' | French: 'S4 256 Row 26 Spare Message French'
  257 = 'Spare' | German: 'S4 257 Row 26 Spare Message German' | French: 'S4 257 Row 26 Spare Message French'
  258 = 'Spare' | German: 'S4 258 Row 26 Spare Message German' | French: 'S4 258 Row 26 Spare Message French'
  259 = 'Spare' | German: 'S4 259 Row 26 Spare Message German' | French: 'S4 259 Row 26 Spare Message French'
  260 = 'Clamp Cylinder A1 Failed to Advance... Check Q1.0...' | German: 'S4 260 Row 27 Failed To Advance.. Check Qxxx.x German' | French: 'S4 260 Row 27 Failed To Advance.. Check Qxxx.x French'
  261 = 'Clamp Cylinder A1 Failed to Return... Check Q1.1...' | German: 'S4 261 Row 27 Failed To Return.. Check Qxxx.x German' | French: 'S4 261 Row 27 Failed To Return.. Check Qxxx.x French'
  262 = 'Clamp Cylinder A1 Lost Advanced... Check I1.0...' | German: 'S4 262 Row 27 Lost Advance Position... Check Ixxx.x German' | French: 'S4 262 Row 27 Lost Advance Position... Check Ixxx.x French'
  263 = 'Clamp Cylinder A1 Lost Returned... Check I1.1...' | German: 'S4 263 Row 27 Lost Return Position... Check Ixxx.x German' | French: 'S4 263 Row 27 Lost Return Position... Check Ixxx.x French'
  264 = 'Clamp Cylinder A1 Switch Fault... Check I1.0, I1.1...' | German: 'S4 264 Row 27 Switch Fault... Check Ixxx.x / Ixxx.x German' | French: 'S4 264 Row 27 Switch Fault... Check Ixxx.x / Ixxx.x French'
  265 = 'Spare' | German: 'S4 265 Row 27 Spare Message German' | French: 'S4 265 Row 27 Spare Message French'
  266 = 'Spare' | German: 'S4 266 Row 27 Spare Message German' | French: 'S4 266 Row 27 Spare Message French'
  267 = 'Spare' | German: 'S4 267 Row 27 Spare Message German' | French: 'S4 267 Row 27 Spare Message French'
  268 = 'Spare' | German: 'S4 268 Row 27 Spare Message German' | French: 'S4 268 Row 27 Spare Message French'
  269 = 'Spare' | German: 'S4 269 Row 27 Spare Message German' | French: 'S4 269 Row 27 Spare Message French'
  270 = 'Clamp Cylinder A1 Failed to Advance... Check Q1.0...' | German: 'S4 270 Row 28 Failed To Advance.. Check Qxxx.x German' | French: 'S4 270 Row 28 Failed To Advance.. Check Qxxx.x French'
  271 = 'Clamp Cylinder A1 Failed to Return... Check Q1.1...' | German: 'S4 271 Row 28 Failed To Return.. Check Qxxx.x German' | French: 'S4 271 Row 28 Failed To Return.. Check Qxxx.x French'
  272 = 'Clamp Cylinder A1 Lost Advanced... Check I1.0...' | German: 'S4 272 Row 28 Lost Advance Position... Check Ixxx.x German' | French: 'S4 272 Row 28 Lost Advance Position... Check Ixxx.x French'
  273 = 'Clamp Cylinder A1 Lost Returned... Check I1.1...' | German: 'S4 273 Row 28 Lost Return Position... Check Ixxx.x German' | French: 'S4 273 Row 28 Lost Return Position... Check Ixxx.x French'
  274 = 'Clamp Cylinder A1 Switch Fault... Check I1.0, I1.1...' | German: 'S4 274 Row 28 Switch Fault... Check Ixxx.x / Ixxx.x German' | French: 'S4 274 Row 28 Switch Fault... Check Ixxx.x / Ixxx.x French'
  275 = 'Spare' | German: 'S4 275 Row 28 Spare Message German' | French: 'S4 275 Row 28 Spare Message French'
  276 = 'Spare' | German: 'S4 276 Row 28 Spare Message German' | French: 'S4 276 Row 28 Spare Message French'
  277 = 'Spare' | German: 'S4 277 Row 28 Spare Message German' | French: 'S4 277 Row 28 Spare Message French'
  278 = 'Spare' | German: 'S4 278 Row 28 Spare Message German' | French: 'S4 278 Row 28 Spare Message French'
  279 = 'Spare' | German: 'S4 279 Row 28 Spare Message German' | French: 'S4 279 Row 28 Spare Message French'
  280 = 'Clamp Cylinder A1 Failed to Advance... Check Q1.0...' | German: 'S4 280 Row 29 Failed To Advance.. Check Qxxx.x German' | French: 'S4 280 Row 29 Failed To Advance.. Check Qxxx.x French'
  281 = 'Clamp Cylinder A1 Failed to Return... Check Q1.1...' | German: 'S4 281 Row 29 Failed To Return.. Check Qxxx.x German' | French: 'S4 281 Row 29 Failed To Return.. Check Qxxx.x French'
  282 = 'Clamp Cylinder A1 Lost Advanced... Check I1.0...' | German: 'S4 282 Row 29 Lost Advance Position... Check Ixxx.x German' | French: 'S4 282 Row 29 Lost Advance Position... Check Ixxx.x French'
  283 = 'Clamp Cylinder A1 Lost Returned... Check I1.1...' | German: 'S4 283 Row 29 Lost Return Position... Check Ixxx.x German' | French: 'S4 283 Row 29 Lost Return Position... Check Ixxx.x French'
  284 = 'Clamp Cylinder A1 Switch Fault... Check I1.0, I1.1...' | German: 'S4 284 Row 29 Switch Fault... Check Ixxx.x / Ixxx.x German' | French: 'S4 284 Row 29 Switch Fault... Check Ixxx.x / Ixxx.x French'
  285 = 'Spare' | German: 'S4 285 Row 29 Spare Message German' | French: 'S4 285 Row 29 Spare Message French'
  286 = 'Spare' | German: 'S4 286 Row 29 Spare Message German' | French: 'S4 286 Row 29 Spare Message French'
  287 = 'Spare' | German: 'S4 287 Row 29 Spare Message German' | French: 'S4 287 Row 29 Spare Message French'
  288 = 'Spare' | German: 'S4 288 Row 29 Spare Message German' | French: 'S4 288 Row 29 Spare Message French'
  289 = 'Spare' | German: 'S4 289 Row 29 Spare Message German' | French: 'S4 289 Row 29 Spare Message French'
  290 = 'Clamp Cylinder A1 Failed to Advance... Check Q1.0...' | German: 'S4 290 Row 30 Failed To Advance.. Check Qxxx.x German' | French: 'S4 290 Row 30 Failed To Advance.. Check Qxxx.x French'
  291 = 'Clamp Cylinder A1 Failed to Return... Check Q1.1...' | German: 'S4 291 Row 30 Failed To Return.. Check Qxxx.x German' | French: 'S4 291 Row 30 Failed To Return.. Check Qxxx.x French'
  292 = 'Clamp Cylinder A1 Lost Advanced... Check I1.0...' | German: 'S4 292 Row 30 Lost Advance Position... Check Ixxx.x German' | French: 'S4 292 Row 30 Lost Advance Position... Check Ixxx.x French'
  293 = 'Clamp Cylinder A1 Lost Returned... Check I1.1...' | German: 'S4 293 Row 30 Lost Return Position... Check Ixxx.x German' | French: 'S4 293 Row 30 Lost Return Position... Check Ixxx.x French'
  294 = 'Clamp Cylinder A1 Switch Fault... Check I1.0, I1.1...' | German: 'S4 294 Row 30 Switch Fault... Check Ixxx.x / Ixxx.x German' | French: 'S4 294 Row 30 Switch Fault... Check Ixxx.x / Ixxx.x French'
  295 = 'Spare' | German: 'S4 295 Row 30 Spare Message German' | French: 'S4 295 Row 30 Spare Message French'
  296 = 'Spare' | German: 'S4 296 Row 30 Spare Message German' | French: 'S4 296 Row 30 Spare Message French'
  297 = 'Spare' | German: 'S4 297 Row 30 Spare Message German' | French: 'S4 297 Row 30 Spare Message French'
  298 = 'Spare' | German: 'S4 298 Row 30 Spare Message German' | French: 'S4 298 Row 30 Spare Message French'
  299 = 'Spare' | German: 'S4 299 Row 30 Spare Message German' | French: 'S4 299 Row 30 Spare Message French'
  300 = 'Clamp Cylinder A1 Failed to Advance... Check Q1.0...' | German: 'S4 300 Row 31 Failed To Advance.. Check Qxxx.x German' | French: 'S4 300 Row 31 Failed To Advance.. Check Qxxx.x French'
  301 = 'Clamp Cylinder A1 Failed to Return... Check Q1.1...' | German: 'S4 301 Row 31 Failed To Return.. Check Qxxx.x German' | French: 'S4 301 Row 31 Failed To Return.. Check Qxxx.x French'
  302 = 'Clamp Cylinder A1 Lost Advanced... Check I1.0...' | German: 'S4 302 Row 31 Lost Advance Position... Check Ixxx.x German' | French: 'S4 302 Row 31 Lost Advance Position... Check Ixxx.x French'
  303 = 'Clamp Cylinder A1 Lost Returned... Check I1.1...' | German: 'S4 303 Row 31 Lost Return Position... Check Ixxx.x German' | French: 'S4 303 Row 31 Lost Return Position... Check Ixxx.x French'
  304 = 'Clamp Cylinder A1 Switch Fault... Check I1.0, I1.1...' | German: 'S4 304 Row 31 Switch Fault... Check Ixxx.x / Ixxx.x German' | French: 'S4 304 Row 31 Switch Fault... Check Ixxx.x / Ixxx.x French'
  305 = 'Spare' | German: 'S4 305 Row 31 Spare Message German' | French: 'S4 305 Row 31 Spare Message French'
  306 = 'Spare' | German: 'S4 306 Row 31 Spare Message German' | French: 'S4 306 Row 31 Spare Message French'
  307 = 'Spare' | German: 'S4 307 Row 31 Spare Message German' | French: 'S4 307 Row 31 Spare Message French'
  308 = 'Spare' | German: 'S4 308 Row 31 Spare Message German' | French: 'S4 308 Row 31 Spare Message French'
  309 = 'Spare' | German: 'S4 309 Row 31 Spare Message German' | French: 'S4 309 Row 31 Spare Message French'
  310 = 'Clamp Cylinder A1 Failed to Advance... Check Q1.0...' | German: 'S4 310 Row 32 Failed To Advance.. Check Qxxx.x German' | French: 'S4 310 Row 32 Failed To Advance.. Check Qxxx.x French'
  311 = 'Clamp Cylinder A1 Failed to Return... Check Q1.1...' | German: 'S4 311 Row 32 Failed To Return.. Check Qxxx.x German' | French: 'S4 311 Row 32 Failed To Return.. Check Qxxx.x French'
  312 = 'Clamp Cylinder A1 Lost Advanced... Check I1.0...' | German: 'S4 312 Row 32 Lost Advance Position... Check Ixxx.x German' | French: 'S4 312 Row 32 Lost Advance Position... Check Ixxx.x French'
  313 = 'Clamp Cylinder A1 Lost Returned... Check I1.1...' | German: 'S4 313 Row 32 Lost Return Position... Check Ixxx.x German' | French: 'S4 313 Row 32 Lost Return Position... Check Ixxx.x French'
  314 = 'Clamp Cylinder A1 Switch Fault... Check I1.0, I1.1...' | German: 'S4 314 Row 32 Switch Fault... Check Ixxx.x / Ixxx.x German' | French: 'S4 314 Row 32 Switch Fault... Check Ixxx.x / Ixxx.x French'
  315 = 'Spare' | German: 'S4 315 Row 32 Spare Message German' | French: 'S4 315 Row 32 Spare Message French'
  316 = 'Spare' | German: 'S4 316 Row 32 Spare Message German' | French: 'S4 316 Row 32 Spare Message French'
  317 = 'Spare' | German: 'S4 317 Row 32 Spare Message German' | French: 'S4 317 Row 32 Spare Message French'
  318 = 'Spare' | German: 'S4 318 Row 32 Spare Message German' | French: 'S4 318 Row 32 Spare Message French'
  319 = 'Spare' | German: 'S4 319 Row 32 Spare Message German' | French: 'S4 319 Row 32 Spare Message French'
  320 = 'Clamp Cylinder A1 Failed to Advance... Check Q1.0...' | German: 'S4 320 Row 33 Failed To Advance.. Check Qxxx.x German' | French: 'S4 320 Row 33 Failed To Advance.. Check Qxxx.x French'
  321 = 'Clamp Cylinder A1 Failed to Return... Check Q1.1...' | German: 'S4 321 Row 33 Failed To Return.. Check Qxxx.x German' | French: 'S4 321 Row 33 Failed To Return.. Check Qxxx.x French'
  322 = 'Clamp Cylinder A1 Lost Advanced... Check I1.0...' | German: 'S4 322 Row 33 Lost Advance Position... Check Ixxx.x German' | French: 'S4 322 Row 33 Lost Advance Position... Check Ixxx.x French'
  323 = 'Clamp Cylinder A1 Lost Returned... Check I1.1...' | German: 'S4 323 Row 33 Lost Return Position... Check Ixxx.x German' | French: 'S4 323 Row 33 Lost Return Position... Check Ixxx.x French'
  324 = 'Clamp Cylinder A1 Switch Fault... Check I1.0, I1.1...' | German: 'S4 324 Row 33 Switch Fault... Check Ixxx.x / Ixxx.x German' | French: 'S4 324 Row 33 Switch Fault... Check Ixxx.x / Ixxx.x French'
  325 = 'Spare' | German: 'S4 325 Row 33 Spare Message German' | French: 'S4 325 Row 33 Spare Message French'
  326 = 'Spare' | German: 'S4 326 Row 33 Spare Message German' | French: 'S4 326 Row 33 Spare Message French'
  327 = 'Spare' | German: 'S4 327 Row 33 Spare Message German' | French: 'S4 327 Row 33 Spare Message French'
  328 = 'Spare' | German: 'S4 328 Row 33 Spare Message German' | French: 'S4 328 Row 33 Spare Message French'
  329 = 'Spare' | German: 'S4 329 Row 33 Spare Message German' | French: 'S4 329 Row 33 Spare Message French'
  330 = 'Clamp Cylinder A1 Failed to Advance... Check Q1.0...' | German: 'S4 330 Row 34 Failed To Advance.. Check Qxxx.x German' | French: 'S4 330 Row 34 Failed To Advance.. Check Qxxx.x French'
  331 = 'Clamp Cylinder A1 Failed to Return... Check Q1.1...' | German: 'S4 331 Row 34 Failed To Return.. Check Qxxx.x German' | French: 'S4 331 Row 34 Failed To Return.. Check Qxxx.x French'
  332 = 'Clamp Cylinder A1 Lost Advanced... Check I1.0...' | German: 'S4 332 Row 34 Lost Advance Position... Check Ixxx.x German' | French: 'S4 332 Row 34 Lost Advance Position... Check Ixxx.x French'
  333 = 'Clamp Cylinder A1 Lost Returned... Check I1.1...' | German: 'S4 333 Row 34 Lost Return Position... Check Ixxx.x German' | French: 'S4 333 Row 34 Lost Return Position... Check Ixxx.x French'
  334 = 'Clamp Cylinder A1 Switch Fault... Check I1.0, I1.1...' | German: 'S4 334 Row 34 Switch Fault... Check Ixxx.x / Ixxx.x German' | French: 'S4 334 Row 34 Switch Fault... Check Ixxx.x / Ixxx.x French'
  335 = 'Spare' | German: 'S4 335 Row 34 Spare Message German' | French: 'S4 335 Row 34 Spare Message French'
  336 = 'Spare' | German: 'S4 336 Row 34 Spare Message German' | French: 'S4 336 Row 34 Spare Message French'
  337 = 'Spare' | German: 'S4 337 Row 34 Spare Message German' | French: 'S4 337 Row 34 Spare Message French'
  338 = 'Spare' | German: 'S4 338 Row 34 Spare Message German' | French: 'S4 338 Row 34 Spare Message French'
  339 = 'Spare' | German: 'S4 339 Row 34 Spare Message German' | French: 'S4 339 Row 34 Spare Message French'
  340 = 'Clamp Cylinder A1 Failed to Advance... Check Q1.0...' | German: 'S4 340 Row 35 Failed To Advance.. Check Qxxx.x German' | French: 'S4 340 Row 35 Failed To Advance.. Check Qxxx.x French'
  341 = 'Clamp Cylinder A1 Failed to Return... Check Q1.1...' | German: 'S4 341 Row 35 Failed To Return.. Check Qxxx.x German' | French: 'S4 341 Row 35 Failed To Return.. Check Qxxx.x French'
  342 = 'Clamp Cylinder A1 Lost Advanced... Check I1.0...' | German: 'S4 342 Row 35 Lost Advance Position... Check Ixxx.x German' | French: 'S4 342 Row 35 Lost Advance Position... Check Ixxx.x French'
  343 = 'Clamp Cylinder A1 Lost Returned... Check I1.1...' | German: 'S4 343 Row 35 Lost Return Position... Check Ixxx.x German' | French: 'S4 343 Row 35 Lost Return Position... Check Ixxx.x French'
  344 = 'Clamp Cylinder A1 Switch Fault... Check I1.0, I1.1...' | German: 'S4 344 Row 35 Switch Fault... Check Ixxx.x / Ixxx.x German' | French: 'S4 344 Row 35 Switch Fault... Check Ixxx.x / Ixxx.x French'
  345 = 'Spare' | German: 'S4 345 Row 35 Spare Message German' | French: 'S4 345 Row 35 Spare Message French'
  346 = 'Spare' | German: 'S4 346 Row 35 Spare Message German' | French: 'S4 346 Row 35 Spare Message French'
  347 = 'Spare' | German: 'S4 347 Row 35 Spare Message German' | French: 'S4 347 Row 35 Spare Message French'
  348 = 'Spare' | German: 'S4 348 Row 35 Spare Message German' | French: 'S4 348 Row 35 Spare Message French'
  349 = 'Spare' | German: 'S4 349 Row 35 Spare Message German' | French: 'S4 349 Row 35 Spare Message French'
  350 = 'Clamp Cylinder A1 Failed to Advance... Check Q1.0...' | German: 'S4 350 Row 36 Failed To Advance.. Check Qxxx.x German' | French: 'S4 350 Row 36 Failed To Advance.. Check Qxxx.x French'
  351 = 'Clamp Cylinder A1 Failed to Return... Check Q1.1...' | German: 'S4 351 Row 36 Failed To Return.. Check Qxxx.x German' | French: 'S4 351 Row 36 Failed To Return.. Check Qxxx.x French'
  352 = 'Clamp Cylinder A1 Lost Advanced... Check I1.0...' | German: 'S4 352 Row 36 Lost Advance Position... Check Ixxx.x German' | French: 'S4 352 Row 36 Lost Advance Position... Check Ixxx.x French'
  353 = 'Clamp Cylinder A1 Lost Returned... Check I1.1...' | German: 'S4 353 Row 36 Lost Return Position... Check Ixxx.x German' | French: 'S4 353 Row 36 Lost Return Position... Check Ixxx.x French'
  354 = 'Clamp Cylinder A1 Switch Fault... Check I1.0, I1.1...' | German: 'S4 354 Row 36 Switch Fault... Check Ixxx.x / Ixxx.x German' | French: 'S4 354 Row 36 Switch Fault... Check Ixxx.x / Ixxx.x French'
  355 = 'Spare' | German: 'S4 355 Row 36 Spare Message German' | French: 'S4 355 Row 36 Spare Message French'
  356 = 'Spare' | German: 'S4 356 Row 36 Spare Message German' | French: 'S4 356 Row 36 Spare Message French'
  357 = 'Spare' | German: 'S4 357 Row 36 Spare Message German' | French: 'S4 357 Row 36 Spare Message French'
  358 = 'Spare' | German: 'S4 358 Row 36 Spare Message German' | French: 'S4 358 Row 36 Spare Message French'
  359 = 'Spare' | German: 'S4 359 Row 36 Spare Message German' | French: 'S4 359 Row 36 Spare Message French'
  360 = 'Clamp Cylinder A1 Failed to Advance... Check Q1.0...' | German: 'S4 360 Row 37 Failed To Advance.. Check Qxxx.x German' | French: 'S4 360 Row 37 Failed To Advance.. Check Qxxx.x French'
  361 = 'Clamp Cylinder A1 Failed to Return... Check Q1.1...' | German: 'S4 361 Row 37 Failed To Return.. Check Qxxx.x German' | French: 'S4 361 Row 37 Failed To Return.. Check Qxxx.x French'
  362 = 'Clamp Cylinder A1 Lost Advanced... Check I1.0...' | German: 'S4 362 Row 37 Lost Advance Position... Check Ixxx.x German' | French: 'S4 362 Row 37 Lost Advance Position... Check Ixxx.x French'
  363 = 'Clamp Cylinder A1 Lost Returned... Check I1.1...' | German: 'S4 363 Row 37 Lost Return Position... Check Ixxx.x German' | French: 'S4 363 Row 37 Lost Return Position... Check Ixxx.x French'
  364 = 'Clamp Cylinder A1 Switch Fault... Check I1.0, I1.1...' | German: 'S4 364 Row 37 Switch Fault... Check Ixxx.x / Ixxx.x German' | French: 'S4 364 Row 37 Switch Fault... Check Ixxx.x / Ixxx.x French'
  365 = 'Spare' | German: 'S4 365 Row 37 Spare Message German' | French: 'S4 365 Row 37 Spare Message French'
  366 = 'Spare' | German: 'S4 366 Row 37 Spare Message German' | French: 'S4 366 Row 37 Spare Message French'
  367 = 'Spare' | German: 'S4 367 Row 37 Spare Message German' | French: 'S4 367 Row 37 Spare Message French'
  368 = 'Spare' | German: 'S4 368 Row 37 Spare Message German' | French: 'S4 368 Row 37 Spare Message French'
  369 = 'Spare' | German: 'S4 369 Row 37 Spare Message German' | French: 'S4 369 Row 37 Spare Message French'
  370 = 'Clamp Cylinder A1 Failed to Advance... Check Q1.0...' | German: 'S4 370 Row 38 Failed To Advance.. Check Qxxx.x German' | French: 'S4 370 Row 38 Failed To Advance.. Check Qxxx.x French'
  371 = 'Clamp Cylinder A1 Failed to Return... Check Q1.1...' | German: 'S4 371 Row 38 Failed To Return.. Check Qxxx.x German' | French: 'S4 371 Row 38 Failed To Return.. Check Qxxx.x French'
  372 = 'Clamp Cylinder A1 Lost Advanced... Check I1.0...' | German: 'S4 372 Row 38 Lost Advance Position... Check Ixxx.x German' | French: 'S4 372 Row 38 Lost Advance Position... Check Ixxx.x French'
  373 = 'Clamp Cylinder A1 Lost Returned... Check I1.1...' | German: 'S4 373 Row 38 Lost Return Position... Check Ixxx.x German' | French: 'S4 373 Row 38 Lost Return Position... Check Ixxx.x French'
  374 = 'Clamp Cylinder A1 Switch Fault... Check I1.0, I1.1...' | German: 'S4 374 Row 38 Switch Fault... Check Ixxx.x / Ixxx.x German' | French: 'S4 374 Row 38 Switch Fault... Check Ixxx.x / Ixxx.x French'
  375 = 'Spare' | German: 'S4 375 Row 38 Spare Message German' | French: 'S4 375 Row 38 Spare Message French'
  376 = 'Spare' | German: 'S4 376 Row 38 Spare Message German' | French: 'S4 376 Row 38 Spare Message French'
  377 = 'Spare' | German: 'S4 377 Row 38 Spare Message German' | French: 'S4 377 Row 38 Spare Message French'
  378 = 'Spare' | German: 'S4 378 Row 38 Spare Message German' | French: 'S4 378 Row 38 Spare Message French'
  379 = 'Spare' | German: 'S4 379 Row 38 Spare Message German' | French: 'S4 379 Row 38 Spare Message French'
  380 = 'Clamp Cylinder A1 Failed to Advance... Check Q1.0...' | German: 'S4 380 Row 39 Failed To Advance.. Check Qxxx.x German' | French: 'S4 380 Row 39 Failed To Advance.. Check Qxxx.x French'
  381 = 'Clamp Cylinder A1 Failed to Return... Check Q1.1...' | German: 'S4 381 Row 39 Failed To Return.. Check Qxxx.x German' | French: 'S4 381 Row 39 Failed To Return.. Check Qxxx.x French'
  382 = 'Clamp Cylinder A1 Lost Advanced... Check I1.0...' | German: 'S4 382 Row 39 Lost Advance Position... Check Ixxx.x German' | French: 'S4 382 Row 39 Lost Advance Position... Check Ixxx.x French'
  383 = 'Clamp Cylinder A1 Lost Returned... Check I1.1...' | German: 'S4 383 Row 39 Lost Return Position... Check Ixxx.x German' | French: 'S4 383 Row 39 Lost Return Position... Check Ixxx.x French'
  384 = 'Clamp Cylinder A1 Switch Fault... Check I1.0, I1.1...' | German: 'S4 384 Row 39 Switch Fault... Check Ixxx.x / Ixxx.x German' | French: 'S4 384 Row 39 Switch Fault... Check Ixxx.x / Ixxx.x French'
  385 = 'Spare' | German: 'S4 385 Row 39 Spare Message German' | French: 'S4 385 Row 39 Spare Message French'
  386 = 'Spare' | German: 'S4 386 Row 39 Spare Message German' | French: 'S4 386 Row 39 Spare Message French'
  387 = 'Spare' | German: 'S4 387 Row 39 Spare Message German' | French: 'S4 387 Row 39 Spare Message French'
  388 = 'Spare' | German: 'S4 388 Row 39 Spare Message German' | French: 'S4 388 Row 39 Spare Message French'
  389 = 'Spare' | German: 'S4 389 Row 39 Spare Message German' | French: 'S4 389 Row 39 Spare Message French'
  390 = 'Clamp Cylinder A1 Failed to Advance... Check Q1.0...' | German: 'S4 390 Row 40 Failed To Advance.. Check Qxxx.x German' | French: 'S4 390 Row 40 Failed To Advance.. Check Qxxx.x French'
  391 = 'Clamp Cylinder A1 Failed to Return... Check Q1.1...' | German: 'S4 391 Row 40 Failed To Return.. Check Qxxx.x German' | French: 'S4 391 Row 40 Failed To Return.. Check Qxxx.x French'
  392 = 'Clamp Cylinder A1 Lost Advanced... Check I1.0...' | German: 'S4 392 Row 40 Lost Advance Position... Check Ixxx.x German' | French: 'S4 392 Row 40 Lost Advance Position... Check Ixxx.x French'
  393 = 'Clamp Cylinder A1 Lost Returned... Check I1.1...' | German: 'S4 393 Row 40 Lost Return Position... Check Ixxx.x German' | French: 'S4 393 Row 40 Lost Return Position... Check Ixxx.x French'
  394 = 'Clamp Cylinder A1 Switch Fault... Check I1.0, I1.1...' | German: 'S4 394 Row 40 Switch Fault... Check Ixxx.x / Ixxx.x German' | French: 'S4 394 Row 40 Switch Fault... Check Ixxx.x / Ixxx.x French'
  395 = 'Spare' | German: 'S4 395 Row 40 Spare Message German' | French: 'S4 395 Row 40 Spare Message French'
  396 = 'Spare' | German: 'S4 396 Row 40 Spare Message German' | French: 'S4 396 Row 40 Spare Message French'
  397 = 'Spare' | German: 'S4 397 Row 40 Spare Message German' | French: 'S4 397 Row 40 Spare Message French'
  398 = 'Spare' | German: 'S4 398 Row 40 Spare Message German' | French: 'S4 398 Row 40 Spare Message French'
  399 = 'Spare' | German: 'S4 399 Row 40 Spare Message German' | French: 'S4 399 Row 40 Spare Message French'
  400 = 'Clamp Cylinder A1 Failed to Advance... Check Q1.0...' | German: 'S4 400 Row 41 Failed To Advance.. Check Qxxx.x German' | French: 'S4 400 Row 41 Failed To Advance.. Check Qxxx.x French'
  401 = 'Clamp Cylinder A1 Failed to Return... Check Q1.1...' | German: 'S4 401 Row 41 Failed To Return.. Check Qxxx.x German' | French: 'S4 401 Row 41 Failed To Return.. Check Qxxx.x French'
  402 = 'Clamp Cylinder A1 Lost Advanced... Check I1.0...' | German: 'S4 402 Row 41 Lost Advance Position... Check Ixxx.x German' | French: 'S4 402 Row 41 Lost Advance Position... Check Ixxx.x French'
  403 = 'Clamp Cylinder A1 Lost Returned... Check I1.1...' | German: 'S4 403 Row 41 Lost Return Position... Check Ixxx.x German' | French: 'S4 403 Row 41 Lost Return Position... Check Ixxx.x French'
  404 = 'Clamp Cylinder A1 Switch Fault... Check I1.0, I1.1...' | German: 'S4 404 Row 41 Switch Fault... Check Ixxx.x / Ixxx.x German' | French: 'S4 404 Row 41 Switch Fault... Check Ixxx.x / Ixxx.x French'
  405 = 'Spare' | German: 'S4 405 Row 41 Spare Message German' | French: 'S4 405 Row 41 Spare Message French'
  406 = 'Spare' | German: 'S4 406 Row 41 Spare Message German' | French: 'S4 406 Row 41 Spare Message French'
  407 = 'Spare' | German: 'S4 407 Row 41 Spare Message German' | French: 'S4 407 Row 41 Spare Message French'
  408 = 'Spare' | German: 'S4 408 Row 41 Spare Message German' | French: 'S4 408 Row 41 Spare Message French'
  409 = 'Spare' | German: 'S4 409 Row 41 Spare Message German' | French: 'S4 409 Row 41 Spare Message French'
  410 = 'Clamp Cylinder A1 Failed to Advance... Check Q1.0...' | German: 'S4 410 Row 42 Failed To Advance.. Check Qxxx.x German' | French: 'S4 410 Row 42 Failed To Advance.. Check Qxxx.x French'
  411 = 'Clamp Cylinder A1 Failed to Return... Check Q1.1...' | German: 'S4 411 Row 42 Failed To Return.. Check Qxxx.x German' | French: 'S4 411 Row 42 Failed To Return.. Check Qxxx.x French'
  412 = 'Clamp Cylinder A1 Lost Advanced... Check I1.0...' | German: 'S4 412 Row 42 Lost Advance Position... Check Ixxx.x German' | French: 'S4 412 Row 42 Lost Advance Position... Check Ixxx.x French'
  413 = 'Clamp Cylinder A1 Lost Returned... Check I1.1...' | German: 'S4 413 Row 42 Lost Return Position... Check Ixxx.x German' | French: 'S4 413 Row 42 Lost Return Position... Check Ixxx.x French'
  414 = 'Clamp Cylinder A1 Switch Fault... Check I1.0, I1.1...' | German: 'S4 414 Row 42 Switch Fault... Check Ixxx.x / Ixxx.x German' | French: 'S4 414 Row 42 Switch Fault... Check Ixxx.x / Ixxx.x French'
  415 = 'Spare' | German: 'S4 415 Row 42 Spare Message German' | French: 'S4 415 Row 42 Spare Message French'
  416 = 'Spare' | German: 'S4 416 Row 42 Spare Message German' | French: 'S4 416 Row 42 Spare Message French'
  417 = 'Spare' | German: 'S4 417 Row 42 Spare Message German' | French: 'S4 417 Row 42 Spare Message French'
  418 = 'Spare' | German: 'S4 418 Row 42 Spare Message German' | French: 'S4 418 Row 42 Spare Message French'
  419 = 'Spare' | German: 'S4 419 Row 42 Spare Message German' | French: 'S4 419 Row 42 Spare Message French'
  420 = 'Clamp Cylinder A1 Failed to Advance... Check Q1.0...' | German: 'S4 420 Row 43 Failed To Advance.. Check Qxxx.x German' | French: 'S4 420 Row 43 Failed To Advance.. Check Qxxx.x French'
  421 = 'Clamp Cylinder A1 Failed to Return... Check Q1.1...' | German: 'S4 421 Row 43 Failed To Return.. Check Qxxx.x German' | French: 'S4 421 Row 43 Failed To Return.. Check Qxxx.x French'
  422 = 'Clamp Cylinder A1 Lost Advanced... Check I1.0...' | German: 'S4 422 Row 43 Lost Advance Position... Check Ixxx.x German' | French: 'S4 422 Row 43 Lost Advance Position... Check Ixxx.x French'
  423 = 'Clamp Cylinder A1 Lost Returned... Check I1.1...' | German: 'S4 423 Row 43 Lost Return Position... Check Ixxx.x German' | French: 'S4 423 Row 43 Lost Return Position... Check Ixxx.x French'
  424 = 'Clamp Cylinder A1 Switch Fault... Check I1.0, I1.1...' | German: 'S4 424 Row 43 Switch Fault... Check Ixxx.x / Ixxx.x German' | French: 'S4 424 Row 43 Switch Fault... Check Ixxx.x / Ixxx.x French'
  425 = 'Spare' | German: 'S4 425 Row 43 Spare Message German' | French: 'S4 425 Row 43 Spare Message French'
  426 = 'Spare' | German: 'S4 426 Row 43 Spare Message German' | French: 'S4 426 Row 43 Spare Message French'
  427 = 'Spare' | German: 'S4 427 Row 43 Spare Message German' | French: 'S4 427 Row 43 Spare Message French'
  428 = 'Spare' | German: 'S4 428 Row 43 Spare Message German' | French: 'S4 428 Row 43 Spare Message French'
  429 = 'Spare' | German: 'S4 429 Row 43 Spare Message German' | French: 'S4 429 Row 43 Spare Message French'
  430 = 'Clamp Cylinder A1 Failed to Advance... Check Q1.0...' | German: 'S4 430 Row 44 Failed To Advance.. Check Qxxx.x German' | French: 'S4 430 Row 44 Failed To Advance.. Check Qxxx.x French'
  431 = 'Clamp Cylinder A1 Failed to Return... Check Q1.1...' | German: 'S4 431 Row 44 Failed To Return.. Check Qxxx.x German' | French: 'S4 431 Row 44 Failed To Return.. Check Qxxx.x French'
  432 = 'Clamp Cylinder A1 Lost Advanced... Check I1.0...' | German: 'S4 432 Row 44 Lost Advance Position... Check Ixxx.x German' | French: 'S4 432 Row 44 Lost Advance Position... Check Ixxx.x French'
  433 = 'Clamp Cylinder A1 Lost Returned... Check I1.1...' | German: 'S4 433 Row 44 Lost Return Position... Check Ixxx.x German' | French: 'S4 433 Row 44 Lost Return Position... Check Ixxx.x French'
  434 = 'Clamp Cylinder A1 Switch Fault... Check I1.0, I1.1...' | German: 'S4 434 Row 44 Switch Fault... Check Ixxx.x / Ixxx.x German' | French: 'S4 434 Row 44 Switch Fault... Check Ixxx.x / Ixxx.x French'
  435 = 'Spare' | German: 'S4 435 Row 44 Spare Message German' | French: 'S4 435 Row 44 Spare Message French'
  436 = 'Spare' | German: 'S4 436 Row 44 Spare Message German' | French: 'S4 436 Row 44 Spare Message French'
  437 = 'Spare' | German: 'S4 437 Row 44 Spare Message German' | French: 'S4 437 Row 44 Spare Message French'
  438 = 'Spare' | German: 'S4 438 Row 44 Spare Message German' | French: 'S4 438 Row 44 Spare Message French'
  439 = 'Spare' | German: 'S4 439 Row 44 Spare Message German' | French: 'S4 439 Row 44 Spare Message French'
  440 = 'Clamp Cylinder A1 Failed to Advance... Check Q1.0...' | German: 'S4 440 Row 45 Failed To Advance.. Check Qxxx.x German' | French: 'S4 440 Row 45 Failed To Advance.. Check Qxxx.x French'
  441 = 'Clamp Cylinder A1 Failed to Return... Check Q1.1...' | German: 'S4 441 Row 45 Failed To Return.. Check Qxxx.x German' | French: 'S4 441 Row 45 Failed To Return.. Check Qxxx.x French'
  442 = 'Clamp Cylinder A1 Lost Advanced... Check I1.0...' | German: 'S4 442 Row 45 Lost Advance Position... Check Ixxx.x German' | French: 'S4 442 Row 45 Lost Advance Position... Check Ixxx.x French'
  443 = 'Clamp Cylinder A1 Lost Returned... Check I1.1...' | German: 'S4 443 Row 45 Lost Return Position... Check Ixxx.x German' | French: 'S4 443 Row 45 Lost Return Position... Check Ixxx.x French'
  444 = 'Clamp Cylinder A1 Switch Fault... Check I1.0, I1.1...' | German: 'S4 444 Row 45 Switch Fault... Check Ixxx.x / Ixxx.x German' | French: 'S4 444 Row 45 Switch Fault... Check Ixxx.x / Ixxx.x French'
  445 = 'Spare' | German: 'S4 445 Row 45 Spare Message German' | French: 'S4 445 Row 45 Spare Message French'
  446 = 'Spare' | German: 'S4 446 Row 45 Spare Message German' | French: 'S4 446 Row 45 Spare Message French'
  447 = 'Spare' | German: 'S4 447 Row 45 Spare Message German' | French: 'S4 447 Row 45 Spare Message French'
  448 = 'Spare' | German: 'S4 448 Row 45 Spare Message German' | French: 'S4 448 Row 45 Spare Message French'
  449 = 'Spare' | German: 'S4 449 Row 45 Spare Message German' | French: 'S4 449 Row 45 Spare Message French'
  450 = 'Clamp Cylinder A1 Failed to Advance... Check Q1.0...' | German: 'S4 450 Row 46 Failed To Advance.. Check Qxxx.x German' | French: 'S4 450 Row 46 Failed To Advance.. Check Qxxx.x French'
  451 = 'Clamp Cylinder A1 Failed to Return... Check Q1.1...' | German: 'S4 451 Row 46 Failed To Return.. Check Qxxx.x German' | French: 'S4 451 Row 46 Failed To Return.. Check Qxxx.x French'
  452 = 'Clamp Cylinder A1 Lost Advanced... Check I1.0...' | German: 'S4 452 Row 46 Lost Advance Position... Check Ixxx.x German' | French: 'S4 452 Row 46 Lost Advance Position... Check Ixxx.x French'
  453 = 'Clamp Cylinder A1 Lost Returned... Check I1.1...' | German: 'S4 453 Row 46 Lost Return Position... Check Ixxx.x German' | French: 'S4 453 Row 46 Lost Return Position... Check Ixxx.x French'
  454 = 'Clamp Cylinder A1 Switch Fault... Check I1.0, I1.1...' | German: 'S4 454 Row 46 Switch Fault... Check Ixxx.x / Ixxx.x German' | French: 'S4 454 Row 46 Switch Fault... Check Ixxx.x / Ixxx.x French'
  455 = 'Spare' | German: 'S4 455 Row 46 Spare Message German' | French: 'S4 455 Row 46 Spare Message French'
  456 = 'Spare' | German: 'S4 456 Row 46 Spare Message German' | French: 'S4 456 Row 46 Spare Message French'
  457 = 'Spare' | German: 'S4 457 Row 46 Spare Message German' | French: 'S4 457 Row 46 Spare Message French'
  458 = 'Spare' | German: 'S4 458 Row 46 Spare Message German' | French: 'S4 458 Row 46 Spare Message French'
  459 = 'Spare' | German: 'S4 459 Row 46 Spare Message German' | French: 'S4 459 Row 46 Spare Message French'
  460 = 'Clamp Cylinder A1 Failed to Advance... Check Q1.0...' | German: 'S4 460 Row 47 Failed To Advance.. Check Qxxx.x German' | French: 'S4 460 Row 47 Failed To Advance.. Check Qxxx.x French'
  461 = 'Clamp Cylinder A1 Failed to Return... Check Q1.1...' | German: 'S4 461 Row 47 Failed To Return.. Check Qxxx.x German' | French: 'S4 461 Row 47 Failed To Return.. Check Qxxx.x French'
  462 = 'Clamp Cylinder A1 Lost Advanced... Check I1.0...' | German: 'S4 462 Row 47 Lost Advance Position... Check Ixxx.x German' | French: 'S4 462 Row 47 Lost Advance Position... Check Ixxx.x French'
  463 = 'Clamp Cylinder A1 Lost Returned... Check I1.1...' | German: 'S4 463 Row 47 Lost Return Position... Check Ixxx.x German' | French: 'S4 463 Row 47 Lost Return Position... Check Ixxx.x French'
  464 = 'Clamp Cylinder A1 Switch Fault... Check I1.0, I1.1...' | German: 'S4 464 Row 47 Switch Fault... Check Ixxx.x / Ixxx.x German' | French: 'S4 464 Row 47 Switch Fault... Check Ixxx.x / Ixxx.x French'
  465 = 'Spare' | German: 'S4 465 Row 47 Spare Message German' | French: 'S4 465 Row 47 Spare Message French'
  466 = 'Spare' | German: 'S4 466 Row 47 Spare Message German' | French: 'S4 466 Row 47 Spare Message French'
  467 = 'Spare' | German: 'S4 467 Row 47 Spare Message German' | French: 'S4 467 Row 47 Spare Message French'
  468 = 'Spare' | German: 'S4 468 Row 47 Spare Message German' | French: 'S4 468 Row 47 Spare Message French'
  469 = 'Spare' | German: 'S4 469 Row 47 Spare Message German' | French: 'S4 469 Row 47 Spare Message French'
  470 = 'Clamp Cylinder A1 Failed to Advance... Check Q1.0...' | German: 'S4 470 Row 48 Failed To Advance.. Check Qxxx.x German' | French: 'S4 470 Row 48 Failed To Advance.. Check Qxxx.x French'
  471 = 'Clamp Cylinder A1 Failed to Return... Check Q1.1...' | German: 'S4 471 Row 48 Failed To Return.. Check Qxxx.x German' | French: 'S4 471 Row 48 Failed To Return.. Check Qxxx.x French'
  472 = 'Clamp Cylinder A1 Lost Advanced... Check I1.0...' | German: 'S4 472 Row 48 Lost Advance Position... Check Ixxx.x German' | French: 'S4 472 Row 48 Lost Advance Position... Check Ixxx.x French'
  473 = 'Clamp Cylinder A1 Lost Returned... Check I1.1...' | German: 'S4 473 Row 48 Lost Return Position... Check Ixxx.x German' | French: 'S4 473 Row 48 Lost Return Position... Check Ixxx.x French'
  474 = 'Clamp Cylinder A1 Switch Fault... Check I1.0, I1.1...' | German: 'S4 474 Row 48 Switch Fault... Check Ixxx.x / Ixxx.x German' | French: 'S4 474 Row 48 Switch Fault... Check Ixxx.x / Ixxx.x French'
  475 = 'Spare' | German: 'S4 475 Row 48 Spare Message German' | French: 'S4 475 Row 48 Spare Message French'
  476 = 'Spare' | German: 'S4 476 Row 48 Spare Message German' | French: 'S4 476 Row 48 Spare Message French'
  477 = 'Spare' | German: 'S4 477 Row 48 Spare Message German' | French: 'S4 477 Row 48 Spare Message French'
  478 = 'Spare' | German: 'S4 478 Row 48 Spare Message German' | French: 'S4 478 Row 48 Spare Message French'
  479 = 'Spare' | German: 'S4 479 Row 48 Spare Message German' | French: 'S4 479 Row 48 Spare Message French'
  480 = 'Clamp Cylinder A1 Failed to Advance... Check Q1.0...' | German: 'S4 480 Row 49 Failed To Advance.. Check Qxxx.x German' | French: 'S4 480 Row 49 Failed To Advance.. Check Qxxx.x French'
  481 = 'Clamp Cylinder A1 Failed to Return... Check Q1.1...' | German: 'S4 481 Row 49 Failed To Return.. Check Qxxx.x German' | French: 'S4 481 Row 49 Failed To Return.. Check Qxxx.x French'
  482 = 'Clamp Cylinder A1 Lost Advanced... Check I1.0...' | German: 'S4 482 Row 49 Lost Advance Position... Check Ixxx.x German' | French: 'S4 482 Row 49 Lost Advance Position... Check Ixxx.x French'
  483 = 'Clamp Cylinder A1 Lost Returned... Check I1.1...' | German: 'S4 483 Row 49 Lost Return Position... Check Ixxx.x German' | French: 'S4 483 Row 49 Lost Return Position... Check Ixxx.x French'
  484 = 'Clamp Cylinder A1 Switch Fault... Check I1.0, I1.1...' | German: 'S4 484 Row 49 Switch Fault... Check Ixxx.x / Ixxx.x German' | French: 'S4 484 Row 49 Switch Fault... Check Ixxx.x / Ixxx.x French'
  485 = 'Spare' | German: 'S4 485 Row 49 Spare Message German' | French: 'S4 485 Row 49 Spare Message French'
  486 = 'Spare' | German: 'S4 486 Row 49 Spare Message German' | French: 'S4 486 Row 49 Spare Message French'
  487 = 'Spare' | German: 'S4 487 Row 49 Spare Message German' | French: 'S4 487 Row 49 Spare Message French'
  488 = 'Spare' | German: 'S4 488 Row 49 Spare Message German' | French: 'S4 488 Row 49 Spare Message French'
  489 = 'Spare' | German: 'S4 489 Row 49 Spare Message German' | French: 'S4 489 Row 49 Spare Message French'
  490 = 'Clamp Cylinder A1 Failed to Advance... Check Q1.0...' | German: 'S4 490 Row 50 Failed To Advance.. Check Qxxx.x German' | French: 'S4 490 Row 50 Failed To Advance.. Check Qxxx.x French'
  491 = 'Clamp Cylinder A1 Failed to Return... Check Q1.1...' | German: 'S4 491 Row 50 Failed To Return.. Check Qxxx.x German' | French: 'S4 491 Row 50 Failed To Return.. Check Qxxx.x French'
  492 = 'Clamp Cylinder A1 Lost Advanced... Check I1.0...' | German: 'S4 492 Row 50 Lost Advance Position... Check Ixxx.x German' | French: 'S4 492 Row 50 Lost Advance Position... Check Ixxx.x French'
  493 = 'Clamp Cylinder A1 Lost Returned... Check I1.1...' | German: 'S4 493 Row 50 Lost Return Position... Check Ixxx.x German' | French: 'S4 493 Row 50 Lost Return Position... Check Ixxx.x French'
  494 = 'Clamp Cylinder A1 Switch Fault... Check I1.0, I1.1...' | German: 'S4 494 Row 50 Switch Fault... Check Ixxx.x / Ixxx.x German' | French: 'S4 494 Row 50 Switch Fault... Check Ixxx.x / Ixxx.x French'
  495 = 'Spare' | German: 'S4 495 Row 50 Spare Message German' | French: 'S4 495 Row 50 Spare Message French'
  496 = 'Spare' | German: 'S4 496 Row 50 Spare Message German' | French: 'S4 496 Row 50 Spare Message French'
  497 = 'Spare' | German: 'S4 497 Row 50 Spare Message German' | French: 'S4 497 Row 50 Spare Message French'
  498 = 'Spare' | German: 'S4 498 Row 50 Spare Message German' | French: 'S4 498 Row 50 Spare Message French'
  499 = 'Spare' | German: 'S4 499 Row 50 Spare Message German' | French: 'S4 499 Row 50 Spare Message French'
  500 = 'Clamp Cylinder A1 Failed to Advance... Check Q1.0...' | German: 'S4 500 Row 51 Failed To Advance.. Check Qxxx.x German' | French: 'S4 500 Row 51 Failed To Advance.. Check Qxxx.x French'
  501 = 'Clamp Cylinder A1 Failed to Return... Check Q1.1...' | German: 'S4 501 Row 51 Failed To Return.. Check Qxxx.x German' | French: 'S4 501 Row 51 Failed To Return.. Check Qxxx.x French'
  502 = 'Clamp Cylinder A1 Lost Advanced... Check I1.0...' | German: 'S4 502 Row 51 Lost Advance Position... Check Ixxx.x German' | French: 'S4 502 Row 51 Lost Advance Position... Check Ixxx.x French'
  503 = 'Clamp Cylinder A1 Lost Returned... Check I1.1...' | German: 'S4 503 Row 51 Lost Return Position... Check Ixxx.x German' | French: 'S4 503 Row 51 Lost Return Position... Check Ixxx.x French'
  504 = 'Clamp Cylinder A1 Switch Fault... Check I1.0, I1.1...' | German: 'S4 504 Row 51 Switch Fault... Check Ixxx.x / Ixxx.x German' | French: 'S4 504 Row 51 Switch Fault... Check Ixxx.x / Ixxx.x French'
  505 = 'Spare' | German: 'S4 505 Row 51 Spare Message German' | French: 'S4 505 Row 51 Spare Message French'
  506 = 'Spare' | German: 'S4 506 Row 51 Spare Message German' | French: 'S4 506 Row 51 Spare Message French'
  507 = 'Spare' | German: 'S4 507 Row 51 Spare Message German' | French: 'S4 507 Row 51 Spare Message French'
  508 = 'Spare' | German: 'S4 508 Row 51 Spare Message German' | French: 'S4 508 Row 51 Spare Message French'
  509 = 'Spare' | German: 'S4 509 Row 51 Spare Message German' | French: 'S4 509 Row 51 Spare Message French'
  510 = 'Clamp Cylinder A1 Failed to Advance... Check Q1.0...' | German: 'S4 510 Row 52 Failed To Advance.. Check Qxxx.x German' | French: 'S4 510 Row 52 Failed To Advance.. Check Qxxx.x French'
  511 = 'Clamp Cylinder A1 Failed to Return... Check Q1.1...' | German: 'S4 511 Row 52 Failed To Return.. Check Qxxx.x German' | French: 'S4 511 Row 52 Failed To Return.. Check Qxxx.x French'
  512 = 'Clamp Cylinder A1 Lost Advanced... Check I1.0...' | German: 'S4 512 Row 52 Lost Advance Position... Check Ixxx.x German' | French: 'S4 512 Row 52 Lost Advance Position... Check Ixxx.x French'
  513 = 'Clamp Cylinder A1 Lost Returned... Check I1.1...' | German: 'S4 513 Row 52 Lost Return Position... Check Ixxx.x German' | French: 'S4 513 Row 52 Lost Return Position... Check Ixxx.x French'
  514 = 'Clamp Cylinder A1 Switch Fault... Check I1.0, I1.1...' | German: 'S4 514 Row 52 Switch Fault... Check Ixxx.x / Ixxx.x German' | French: 'S4 514 Row 52 Switch Fault... Check Ixxx.x / Ixxx.x French'
  515 = 'Spare' | German: 'S4 515 Row 52 Spare Message German' | French: 'S4 515 Row 52 Spare Message French'
  516 = 'Spare' | German: 'S4 516 Row 52 Spare Message German' | French: 'S4 516 Row 52 Spare Message French'
  517 = 'Spare' | German: 'S4 517 Row 52 Spare Message German' | French: 'S4 517 Row 52 Spare Message French'
  518 = 'Spare' | German: 'S4 518 Row 52 Spare Message German' | French: 'S4 518 Row 52 Spare Message French'
  519 = 'Spare' | German: 'S4 519 Row 52 Spare Message German' | French: 'S4 519 Row 52 Spare Message French'
  520 = 'Clamp Cylinder A1 Failed to Advance... Check Q1.0...' | German: 'S4 520 Row 53 Failed To Advance.. Check Qxxx.x German' | French: 'S4 520 Row 53 Failed To Advance.. Check Qxxx.x French'
  521 = 'Clamp Cylinder A1 Failed to Return... Check Q1.1...' | German: 'S4 521 Row 53 Failed To Return.. Check Qxxx.x German' | French: 'S4 521 Row 53 Failed To Return.. Check Qxxx.x French'
  522 = 'Clamp Cylinder A1 Lost Advanced... Check I1.0...' | German: 'S4 522 Row 53 Lost Advance Position... Check Ixxx.x German' | French: 'S4 522 Row 53 Lost Advance Position... Check Ixxx.x French'
  523 = 'Clamp Cylinder A1 Lost Returned... Check I1.1...' | German: 'S4 523 Row 53 Lost Return Position... Check Ixxx.x German' | French: 'S4 523 Row 53 Lost Return Position... Check Ixxx.x French'
  524 = 'Clamp Cylinder A1 Switch Fault... Check I1.0, I1.1...' | German: 'S4 524 Row 53 Switch Fault... Check Ixxx.x / Ixxx.x German' | French: 'S4 524 Row 53 Switch Fault... Check Ixxx.x / Ixxx.x French'
  525 = 'Spare' | German: 'S4 525 Row 53 Spare Message German' | French: 'S4 525 Row 53 Spare Message French'
  526 = 'Spare' | German: 'S4 526 Row 53 Spare Message German' | French: 'S4 526 Row 53 Spare Message French'
  527 = 'Spare' | German: 'S4 527 Row 53 Spare Message German' | French: 'S4 527 Row 53 Spare Message French'
  528 = 'Spare' | German: 'S4 528 Row 53 Spare Message German' | French: 'S4 528 Row 53 Spare Message French'
  529 = 'Spare' | German: 'S4 529 Row 53 Spare Message German' | French: 'S4 529 Row 53 Spare Message French'
  530 = 'Clamp Cylinder A1 Failed to Advance... Check Q1.0...' | German: 'S4 530 Row 54 Failed To Advance.. Check Qxxx.x German' | French: 'S4 530 Row 54 Failed To Advance.. Check Qxxx.x French'
  531 = 'Clamp Cylinder A1 Failed to Return... Check Q1.1...' | German: 'S4 531 Row 54 Failed To Return.. Check Qxxx.x German' | French: 'S4 531 Row 54 Failed To Return.. Check Qxxx.x French'
  532 = 'Clamp Cylinder A1 Lost Advanced... Check I1.0...' | German: 'S4 532 Row 54 Lost Advance Position... Check Ixxx.x German' | French: 'S4 532 Row 54 Lost Advance Position... Check Ixxx.x French'
  533 = 'Clamp Cylinder A1 Lost Returned... Check I1.1...' | German: 'S4 533 Row 54 Lost Return Position... Check Ixxx.x German' | French: 'S4 533 Row 54 Lost Return Position... Check Ixxx.x French'
  534 = 'Clamp Cylinder A1 Switch Fault... Check I1.0, I1.1...' | German: 'S4 534 Row 54 Switch Fault... Check Ixxx.x / Ixxx.x German' | French: 'S4 534 Row 54 Switch Fault... Check Ixxx.x / Ixxx.x French'
  535 = 'Spare' | German: 'S4 535 Row 54 Spare Message German' | French: 'S4 535 Row 54 Spare Message French'
  536 = 'Spare' | German: 'S4 536 Row 54 Spare Message German' | French: 'S4 536 Row 54 Spare Message French'
  537 = 'Spare' | German: 'S4 537 Row 54 Spare Message German' | French: 'S4 537 Row 54 Spare Message French'
  538 = 'Spare' | German: 'S4 538 Row 54 Spare Message German' | French: 'S4 538 Row 54 Spare Message French'
  539 = 'Spare' | German: 'S4 539 Row 54 Spare Message German' | French: 'S4 539 Row 54 Spare Message French'
  540 = 'Clamp Cylinder A1 Failed to Advance... Check Q1.0...' | German: 'S4 540 Row 55 Failed To Advance.. Check Qxxx.x German' | French: 'S4 540 Row 55 Failed To Advance.. Check Qxxx.x French'
  541 = 'Clamp Cylinder A1 Failed to Return... Check Q1.1...' | German: 'S4 541 Row 55 Failed To Return.. Check Qxxx.x German' | French: 'S4 541 Row 55 Failed To Return.. Check Qxxx.x French'
  542 = 'Clamp Cylinder A1 Lost Advanced... Check I1.0...' | German: 'S4 542 Row 55 Lost Advance Position... Check Ixxx.x German' | French: 'S4 542 Row 55 Lost Advance Position... Check Ixxx.x French'
  543 = 'Clamp Cylinder A1 Lost Returned... Check I1.1...' | German: 'S4 543 Row 55 Lost Return Position... Check Ixxx.x German' | French: 'S4 543 Row 55 Lost Return Position... Check Ixxx.x French'
  544 = 'Clamp Cylinder A1 Switch Fault... Check I1.0, I1.1...' | German: 'S4 544 Row 55 Switch Fault... Check Ixxx.x / Ixxx.x German' | French: 'S4 544 Row 55 Switch Fault... Check Ixxx.x / Ixxx.x French'
  545 = 'Spare' | German: 'S4 545 Row 55 Spare Message German' | French: 'S4 545 Row 55 Spare Message French'
  546 = 'Spare' | German: 'S4 546 Row 55 Spare Message German' | French: 'S4 546 Row 55 Spare Message French'
  547 = 'Spare' | German: 'S4 547 Row 55 Spare Message German' | French: 'S4 547 Row 55 Spare Message French'
  548 = 'Spare' | German: 'S4 548 Row 55 Spare Message German' | French: 'S4 548 Row 55 Spare Message French'
  549 = 'Spare' | German: 'S4 549 Row 55 Spare Message German' | French: 'S4 549 Row 55 Spare Message French'
  550 = 'Clamp Cylinder A1 Failed to Advance... Check Q1.0...' | German: 'S4 550 Row 56 Failed To Advance.. Check Qxxx.x German' | French: 'S4 550 Row 56 Failed To Advance.. Check Qxxx.x French'
  551 = 'Clamp Cylinder A1 Failed to Return... Check Q1.1...' | German: 'S4 551 Row 56 Failed To Return.. Check Qxxx.x German' | French: 'S4 551 Row 56 Failed To Return.. Check Qxxx.x French'
  552 = 'Clamp Cylinder A1 Lost Advanced... Check I1.0...' | German: 'S4 552 Row 56 Lost Advance Position... Check Ixxx.x German' | French: 'S4 552 Row 56 Lost Advance Position... Check Ixxx.x French'
  553 = 'Clamp Cylinder A1 Lost Returned... Check I1.1...' | German: 'S4 553 Row 56 Lost Return Position... Check Ixxx.x German' | French: 'S4 553 Row 56 Lost Return Position... Check Ixxx.x French'
  554 = 'Clamp Cylinder A1 Switch Fault... Check I1.0, I1.1...' | German: 'S4 554 Row 56 Switch Fault... Check Ixxx.x / Ixxx.x German' | French: 'S4 554 Row 56 Switch Fault... Check Ixxx.x / Ixxx.x French'
  555 = 'Spare' | German: 'S4 555 Row 56 Spare Message German' | French: 'S4 555 Row 56 Spare Message French'
  556 = 'Spare' | German: 'S4 556 Row 56 Spare Message German' | French: 'S4 556 Row 56 Spare Message French'
  557 = 'Spare' | German: 'S4 557 Row 56 Spare Message German' | French: 'S4 557 Row 56 Spare Message French'
  558 = 'Spare' | German: 'S4 558 Row 56 Spare Message German' | French: 'S4 558 Row 56 Spare Message French'
  559 = 'Spare' | German: 'S4 559 Row 56 Spare Message German' | French: 'S4 559 Row 56 Spare Message French'
  560 = 'Clamp Cylinder A1 Failed to Advance... Check Q1.0...' | German: 'S4 560 Row 57 Failed To Advance.. Check Qxxx.x German' | French: 'S4 560 Row 57 Failed To Advance.. Check Qxxx.x French'
  561 = 'Clamp Cylinder A1 Failed to Return... Check Q1.1...' | German: 'S4 561 Row 57 Failed To Return.. Check Qxxx.x German' | French: 'S4 561 Row 57 Failed To Return.. Check Qxxx.x French'
  562 = 'Clamp Cylinder A1 Lost Advanced... Check I1.0...' | German: 'S4 562 Row 57 Lost Advance Position... Check Ixxx.x German' | French: 'S4 562 Row 57 Lost Advance Position... Check Ixxx.x French'
  563 = 'Clamp Cylinder A1 Lost Returned... Check I1.1...' | German: 'S4 563 Row 57 Lost Return Position... Check Ixxx.x German' | French: 'S4 563 Row 57 Lost Return Position... Check Ixxx.x French'
  564 = 'Clamp Cylinder A1 Switch Fault... Check I1.0, I1.1...' | German: 'S4 564 Row 57 Switch Fault... Check Ixxx.x / Ixxx.x German' | French: 'S4 564 Row 57 Switch Fault... Check Ixxx.x / Ixxx.x French'
  565 = 'Spare' | German: 'S4 565 Row 57 Spare Message German' | French: 'S4 565 Row 57 Spare Message French'
  566 = 'Spare' | German: 'S4 566 Row 57 Spare Message German' | French: 'S4 566 Row 57 Spare Message French'
  567 = 'Spare' | German: 'S4 567 Row 57 Spare Message German' | French: 'S4 567 Row 57 Spare Message French'
  568 = 'Spare' | German: 'S4 568 Row 57 Spare Message German' | French: 'S4 568 Row 57 Spare Message French'
  569 = 'Spare' | German: 'S4 569 Row 57 Spare Message German' | French: 'S4 569 Row 57 Spare Message French'
  570 = 'Clamp Cylinder A1 Failed to Advance... Check Q1.0...' | German: 'S4 570 Row 58 Failed To Advance.. Check Qxxx.x German' | French: 'S4 570 Row 58 Failed To Advance.. Check Qxxx.x French'
  571 = 'Clamp Cylinder A1 Failed to Return... Check Q1.1...' | German: 'S4 571 Row 58 Failed To Return.. Check Qxxx.x German' | French: 'S4 571 Row 58 Failed To Return.. Check Qxxx.x French'
  572 = 'Clamp Cylinder A1 Lost Advanced... Check I1.0...' | German: 'S4 572 Row 58 Lost Advance Position... Check Ixxx.x German' | French: 'S4 572 Row 58 Lost Advance Position... Check Ixxx.x French'
  573 = 'Clamp Cylinder A1 Lost Returned... Check I1.1...' | German: 'S4 573 Row 58 Lost Return Position... Check Ixxx.x German' | French: 'S4 573 Row 58 Lost Return Position... Check Ixxx.x French'
  574 = 'Clamp Cylinder A1 Switch Fault... Check I1.0, I1.1...' | German: 'S4 574 Row 58 Switch Fault... Check Ixxx.x / Ixxx.x German' | French: 'S4 574 Row 58 Switch Fault... Check Ixxx.x / Ixxx.x French'
  575 = 'Spare' | German: 'S4 575 Row 58 Spare Message German' | French: 'S4 575 Row 58 Spare Message French'
  576 = 'Spare' | German: 'S4 576 Row 58 Spare Message German' | French: 'S4 576 Row 58 Spare Message French'
  577 = 'Spare' | German: 'S4 577 Row 58 Spare Message German' | French: 'S4 577 Row 58 Spare Message French'
  578 = 'Spare' | German: 'S4 578 Row 58 Spare Message German' | French: 'S4 578 Row 58 Spare Message French'
  579 = 'Spare' | German: 'S4 579 Row 58 Spare Message German' | French: 'S4 579 Row 58 Spare Message French'
  580 = 'Clamp Cylinder A1 Failed to Advance... Check Q1.0...' | German: 'S4 580 Row 59 Failed To Advance.. Check Qxxx.x German' | French: 'S4 580 Row 59 Failed To Advance.. Check Qxxx.x French'
  581 = 'Clamp Cylinder A1 Failed to Return... Check Q1.1...' | German: 'S4 581 Row 59 Failed To Return.. Check Qxxx.x German' | French: 'S4 581 Row 59 Failed To Return.. Check Qxxx.x French'
  582 = 'Clamp Cylinder A1 Lost Advanced... Check I1.0...' | German: 'S4 582 Row 59 Lost Advance Position... Check Ixxx.x German' | French: 'S4 582 Row 59 Lost Advance Position... Check Ixxx.x French'
  583 = 'Clamp Cylinder A1 Lost Returned... Check I1.1...' | German: 'S4 583 Row 59 Lost Return Position... Check Ixxx.x German' | French: 'S4 583 Row 59 Lost Return Position... Check Ixxx.x French'
  584 = 'Clamp Cylinder A1 Switch Fault... Check I1.0, I1.1...' | German: 'S4 584 Row 59 Switch Fault... Check Ixxx.x / Ixxx.x German' | French: 'S4 584 Row 59 Switch Fault... Check Ixxx.x / Ixxx.x French'
  585 = 'Spare' | German: 'S4 585 Row 59 Spare Message German' | French: 'S4 585 Row 59 Spare Message French'
  586 = 'Spare' | German: 'S4 586 Row 59 Spare Message German' | French: 'S4 586 Row 59 Spare Message French'
  587 = 'Spare' | German: 'S4 587 Row 59 Spare Message German' | French: 'S4 587 Row 59 Spare Message French'
  588 = 'Spare' | German: 'S4 588 Row 59 Spare Message German' | French: 'S4 588 Row 59 Spare Message French'
  589 = 'Spare' | German: 'S4 589 Row 59 Spare Message German' | French: 'S4 589 Row 59 Spare Message French'
  590 = 'Clamp Cylinder A1 Failed to Advance... Check Q1.0...' | German: 'S4 590 Row 60 Failed To Advance.. Check Qxxx.x German' | French: 'S4 590 Row 60 Failed To Advance.. Check Qxxx.x French'
  591 = 'Clamp Cylinder A1 Failed to Return... Check Q1.1...' | German: 'S4 591 Row 60 Failed To Return.. Check Qxxx.x German' | French: 'S4 591 Row 60 Failed To Return.. Check Qxxx.x French'
  592 = 'Clamp Cylinder A1 Lost Advanced... Check I1.0...' | German: 'S4 592 Row 60 Lost Advance Position... Check Ixxx.x German' | French: 'S4 592 Row 60 Lost Advance Position... Check Ixxx.x French'
  593 = 'Clamp Cylinder A1 Lost Returned... Check I1.1...' | German: 'S4 593 Row 60 Lost Return Position... Check Ixxx.x German' | French: 'S4 593 Row 60 Lost Return Position... Check Ixxx.x French'
  594 = 'Clamp Cylinder A1 Switch Fault... Check I1.0, I1.1...' | German: 'S4 594 Row 60 Switch Fault... Check Ixxx.x / Ixxx.x German' | French: 'S4 594 Row 60 Switch Fault... Check Ixxx.x / Ixxx.x French'
  595 = 'Spare' | German: 'S4 595 Row 60 Spare Message German' | French: 'S4 595 Row 60 Spare Message French'
  596 = 'Spare' | German: 'S4 596 Row 60 Spare Message German' | French: 'S4 596 Row 60 Spare Message French'
  597 = 'Spare' | German: 'S4 597 Row 60 Spare Message German' | French: 'S4 597 Row 60 Spare Message French'
  598 = 'Spare' | German: 'S4 598 Row 60 Spare Message German' | French: 'S4 598 Row 60 Spare Message French'
  599 = 'Spare' | German: 'S4 599 Row 60 Spare Message German' | French: 'S4 599 Row 60 Spare Message French'
  600 = 'Clamp Cylinder A1 Failed to Advance... Check Q1.0...' | German: 'S4 600 Row 61 Failed To Advance.. Check Qxxx.x German' | French: 'S4 600 Row 61 Failed To Advance.. Check Qxxx.x French'
  601 = 'Clamp Cylinder A1 Failed to Return... Check Q1.1...' | German: 'S4 601 Row 61 Failed To Return.. Check Qxxx.x German' | French: 'S4 601 Row 61 Failed To Return.. Check Qxxx.x French'
  602 = 'Clamp Cylinder A1 Lost Advanced... Check I1.0...' | German: 'S4 602 Row 61 Lost Advance Position... Check Ixxx.x German' | French: 'S4 602 Row 61 Lost Advance Position... Check Ixxx.x French'
  603 = 'Clamp Cylinder A1 Lost Returned... Check I1.1...' | German: 'S4 603 Row 61 Lost Return Position... Check Ixxx.x German' | French: 'S4 603 Row 61 Lost Return Position... Check Ixxx.x French'
  604 = 'Clamp Cylinder A1 Switch Fault... Check I1.0, I1.1...' | German: 'S4 604 Row 61 Switch Fault... Check Ixxx.x / Ixxx.x German' | French: 'S4 604 Row 61 Switch Fault... Check Ixxx.x / Ixxx.x French'
  605 = 'Spare' | German: 'S4 605 Row 61 Spare Message German' | French: 'S4 605 Row 61 Spare Message French'
  606 = 'Spare' | German: 'S4 606 Row 61 Spare Message German' | French: 'S4 606 Row 61 Spare Message French'
  607 = 'Spare' | German: 'S4 607 Row 61 Spare Message German' | French: 'S4 607 Row 61 Spare Message French'
  608 = 'Spare' | German: 'S4 608 Row 61 Spare Message German' | French: 'S4 608 Row 61 Spare Message French'
  609 = 'Spare' | German: 'S4 609 Row 61 Spare Message German' | French: 'S4 609 Row 61 Spare Message French'
  610 = 'Clamp Cylinder A1 Failed to Advance... Check Q1.0...' | German: 'S4 610 Row 62 Failed To Advance.. Check Qxxx.x German' | French: 'S4 610 Row 62 Failed To Advance.. Check Qxxx.x French'
  611 = 'Clamp Cylinder A1 Failed to Return... Check Q1.1...' | German: 'S4 611 Row 62 Failed To Return.. Check Qxxx.x German' | French: 'S4 611 Row 62 Failed To Return.. Check Qxxx.x French'
  612 = 'Clamp Cylinder A1 Lost Advanced... Check I1.0...' | German: 'S4 612 Row 62 Lost Advance Position... Check Ixxx.x German' | French: 'S4 612 Row 62 Lost Advance Position... Check Ixxx.x French'
  613 = 'Clamp Cylinder A1 Lost Returned... Check I1.1...' | German: 'S4 613 Row 62 Lost Return Position... Check Ixxx.x German' | French: 'S4 613 Row 62 Lost Return Position... Check Ixxx.x French'
  614 = 'Clamp Cylinder A1 Switch Fault... Check I1.0, I1.1...' | German: 'S4 614 Row 62 Switch Fault... Check Ixxx.x / Ixxx.x German' | French: 'S4 614 Row 62 Switch Fault... Check Ixxx.x / Ixxx.x French'
  615 = 'Spare' | German: 'S4 615 Row 62 Spare Message German' | French: 'S4 615 Row 62 Spare Message French'
  616 = 'Spare' | German: 'S4 616 Row 62 Spare Message German' | French: 'S4 616 Row 62 Spare Message French'
  617 = 'Spare' | German: 'S4 617 Row 62 Spare Message German' | French: 'S4 617 Row 62 Spare Message French'
  618 = 'Spare' | German: 'S4 618 Row 62 Spare Message German' | French: 'S4 618 Row 62 Spare Message French'
  619 = 'Spare' | German: 'S4 619 Row 62 Spare Message German' | French: 'S4 619 Row 62 Spare Message French'
  620 = 'Clamp Cylinder A1 Failed to Advance... Check Q1.0...' | German: 'S4 620 Row 63 Failed To Advance.. Check Qxxx.x German' | French: 'S4 620 Row 63 Failed To Advance.. Check Qxxx.x French'
  621 = 'Clamp Cylinder A1 Failed to Return... Check Q1.1...' | German: 'S4 621 Row 63 Failed To Return.. Check Qxxx.x German' | French: 'S4 621 Row 63 Failed To Return.. Check Qxxx.x French'
  622 = 'Clamp Cylinder A1 Lost Advanced... Check I1.0...' | German: 'S4 622 Row 63 Lost Advance Position... Check Ixxx.x German' | French: 'S4 622 Row 63 Lost Advance Position... Check Ixxx.x French'
  623 = 'Clamp Cylinder A1 Lost Returned... Check I1.1...' | German: 'S4 623 Row 63 Lost Return Position... Check Ixxx.x German' | French: 'S4 623 Row 63 Lost Return Position... Check Ixxx.x French'
  624 = 'Clamp Cylinder A1 Switch Fault... Check I1.0, I1.1...' | German: 'S4 624 Row 63 Switch Fault... Check Ixxx.x / Ixxx.x German' | French: 'S4 624 Row 63 Switch Fault... Check Ixxx.x / Ixxx.x French'
  625 = 'Spare' | German: 'S4 625 Row 63 Spare Message German' | French: 'S4 625 Row 63 Spare Message French'
  626 = 'Spare' | German: 'S4 626 Row 63 Spare Message German' | French: 'S4 626 Row 63 Spare Message French'
  627 = 'Spare' | German: 'S4 627 Row 63 Spare Message German' | French: 'S4 627 Row 63 Spare Message French'
  628 = 'Spare' | German: 'S4 628 Row 63 Spare Message German' | French: 'S4 628 Row 63 Spare Message French'
  629 = 'Spare' | German: 'S4 629 Row 63 Spare Message German' | French: 'S4 629 Row 63 Spare Message French'
  630 = 'Clamp Cylinder A1 Failed to Advance... Check Q1.0...' | German: 'S4 630 Row 64 Failed To Advance.. Check Qxxx.x German' | French: 'S4 630 Row 64 Failed To Advance.. Check Qxxx.x French'
  631 = 'Clamp Cylinder A1 Failed to Return... Check Q1.1...' | German: 'S4 631 Row 64 Failed To Return.. Check Qxxx.x German' | French: 'S4 631 Row 64 Failed To Return.. Check Qxxx.x French'
  632 = 'Clamp Cylinder A1 Lost Advanced... Check I1.0...' | German: 'S4 632 Row 64 Lost Advance Position... Check Ixxx.x German' | French: 'S4 632 Row 64 Lost Advance Position... Check Ixxx.x French'
  633 = 'Clamp Cylinder A1 Lost Returned... Check I1.1...' | German: 'S4 633 Row 64 Lost Return Position... Check Ixxx.x German' | French: 'S4 633 Row 64 Lost Return Position... Check Ixxx.x French'
  634 = 'Clamp Cylinder A1 Switch Fault... Check I1.0, I1.1...' | German: 'S4 634 Row 64 Switch Fault... Check Ixxx.x / Ixxx.x German' | French: 'S4 634 Row 64 Switch Fault... Check Ixxx.x / Ixxx.x French'
  635 = 'Spare' | German: 'S4 635 Row 64 Spare Message German' | French: 'S4 635 Row 64 Spare Message French'
  636 = 'Spare' | German: 'S4 636 Row 64 Spare Message German' | French: 'S4 636 Row 64 Spare Message French'
  637 = 'Spare' | German: 'S4 637 Row 64 Spare Message German' | French: 'S4 637 Row 64 Spare Message French'
  638 = 'Spare' | German: 'S4 638 Row 64 Spare Message German' | French: 'S4 638 Row 64 Spare Message French'
  639 = 'Spare' | German: 'S4 639 Row 64 Spare Message German' | French: 'S4 639 Row 64 Spare Message French'
  640 = 'Clamp Cylinder A1 Failed to Advance... Check Q1.0...' | German: 'S4 640 Row 65 Failed To Advance.. Check Qxxx.x German' | French: 'S4 640 Row 65 Failed To Advance.. Check Qxxx.x French'
  641 = 'Clamp Cylinder A1 Failed to Return... Check Q1.1...' | German: 'S4 641 Row 65 Failed To Return.. Check Qxxx.x German' | French: 'S4 641 Row 65 Failed To Return.. Check Qxxx.x French'
  642 = 'Clamp Cylinder A1 Lost Advanced... Check I1.0...' | German: 'S4 642 Row 65 Lost Advance Position... Check Ixxx.x German' | French: 'S4 642 Row 65 Lost Advance Position... Check Ixxx.x French'
  643 = 'Clamp Cylinder A1 Lost Returned... Check I1.1...' | German: 'S4 643 Row 65 Lost Return Position... Check Ixxx.x German' | French: 'S4 643 Row 65 Lost Return Position... Check Ixxx.x French'
  644 = 'Clamp Cylinder A1 Switch Fault... Check I1.0, I1.1...' | German: 'S4 644 Row 65 Switch Fault... Check Ixxx.x / Ixxx.x German' | French: 'S4 644 Row 65 Switch Fault... Check Ixxx.x / Ixxx.x French'
  645 = 'Spare' | German: 'S4 645 Row 65 Spare Message German' | French: 'S4 645 Row 65 Spare Message French'
  646 = 'Spare' | German: 'S4 646 Row 65 Spare Message German' | French: 'S4 646 Row 65 Spare Message French'
  647 = 'Spare' | German: 'S4 647 Row 65 Spare Message German' | French: 'S4 647 Row 65 Spare Message French'
  648 = 'Spare' | German: 'S4 648 Row 65 Spare Message German' | French: 'S4 648 Row 65 Spare Message French'
  649 = 'Spare' | German: 'S4 649 Row 65 Spare Message German' | French: 'S4 649 Row 65 Spare Message French'
